// TwinCAT 3 PLC project Untitled1
// ProgramVersion: 3.1.4023.0
// libraries:
//   CmpBitmapPool, * (System)
//   Tc2_SerialCom, * (Beckhoff Automation GmbH)
//   Tc2_Standard, * (Beckhoff Automation GmbH)
//   Tc2_SUPS, * (Beckhoff Automation GmbH)
//   Tc2_System, * (Beckhoff Automation GmbH)
//   Tc2_Utilities, * (Beckhoff Automation GmbH)
//   Tc3_Module, * (Beckhoff Automation GmbH)
//   VisuDialogs, * (System)
//   VisuSymbols,3.5.10.0,System
// project tree:
//   01. MAIN/01.1 ReactorTemperature/DUTs/ ST_PidParameters.TcDUT
//   01. MAIN/01.1 ReactorTemperature/FBs/ FB_PidControllerRelayOutput.TcPOU, FB_ReactorTemperatureControlStateMachine.TcPOU (not stored)
//   01. MAIN/01.1 ReactorTemperature/Handlers/01.1.1 TemperatureSensorScaling/ TemperatureSensorScalingHandler.TcPOU
//   01. MAIN/01.1 ReactorTemperature/Handlers/01.1.2 ReactorTemperatureControl/ ReactorTemperatureControlHandler.TcPOU
//   01. MAIN/01.1 ReactorTemperature/ ReactorTemperatureController.TcPOU
//   01. MAIN/01.2 ReactorLevelAndPressure/DUTs/ E_AutomaticExtractionState.TcDUT (not stored), ST_AutomaticExtractionParameters.TcDUT (not stored), ST_AutomaticExtractionValues.TcDUT, ST_ExtractiveControlValveCommands.TcDUT, ST_ExtractiveControlValveParameters.TcDUT, ST_ExtractiveOnOffValveValues.TcDUT (not stored), ST_PressureIntervals.TcDUT (not stored)
//   01. MAIN/01.2 ReactorLevelAndPressure/FBs/ FB_AutomaticExtractionStateMachine.TcPOU, FB_ControlValveStateMachine.TcPOU, FB_ExtractiveOutletControl.TcPOU, FB_ReactorValves.TcPOU, FB_Runtime.TcPOU, FB_ValveTrigger.TcPOU (not stored), F_RoundToClosest.TcPOU (not stored)
//   01. MAIN/01.2 ReactorLevelAndPressure/Handlers/01.2.1 PressureSensorScaling/ PressureSensorScalingHandler.TcPOU
//   01. MAIN/01.2 ReactorLevelAndPressure/Handlers/01.2.2 AutomaticExtraction/ AutomaticExtractionHandler.TcPOU
//   01. MAIN/01.2 ReactorLevelAndPressure/Handlers/01.2.3 ExtractiveOutlet/ ExtractiveOutletHandler.TcPOU
//   01. MAIN/01.2 ReactorLevelAndPressure/ ReactorLevelAndPressureController.TcPOU
//   01. MAIN/01.3 ReactorFlow/DUTs/ ST_FlowControlCommands.TcDUT, ST_FlowControlParameters.TcDUT, ST_MPC_Matrices.TcDUT
//   01. MAIN/01.3 ReactorFlow/FBs/ FB_ConsumptionCalculator.TcPOU, FB_mF.TcPOU, FB_MovingAverage.TcPOU, FB_MPC.TcPOU
//   01. MAIN/01.3 ReactorFlow/Handlers/01.3.1 Co2MeanFlowCalculation/ FB_Co2MeanFlowCalculationHandler.TcPOU
//   01. MAIN/01.3 ReactorFlow/Handlers/01.3.2 Co2Consumption/ FB_Co2ConsumptionHandler.TcPOU
//   01. MAIN/01.3 ReactorFlow/Handlers/01.3.3 Co2FlowModeling/ FB_Co2FlowModelingHandler.TcPOU
//   01. MAIN/01.3 ReactorFlow/Handlers/01.3.4 Co2FlowModelDeviation/ FB_Co2FlowModelDeviationHandler.TcPOU
//   01. MAIN/01.3 ReactorFlow/Handlers/01.3.5 FlowMpc/ FB_FlowMpcHandler.TcPOU
//   01. MAIN/01.3 ReactorFlow/ ReactorFlowController.TcPOU
//   01. MAIN/01.4 DataAcquisition/ DataAcquisitionController.TcPOU
//   01. MAIN/01.4 DataAcquisition/DUTs/ ST_MatlabValues.TcDUT (not stored)
//   01. MAIN/01.4 DataAcquisition/FBs/ FB_HeartBeat.TcPOU
//   01. MAIN/01.4 DataAcquisition/Handlers/01.4.1 OpcTagWriting/ OpcTagWritingHandler.TcPOU
//   01. MAIN/01.4 DataAcquisition/Handlers/01.4.2 Matlab/ MatlabHandler.TcPOU (not stored)
//   01. MAIN/01.4 DataAcquisition/Handlers/01.4.3 SpecialDataWriting/ SpecialDataWritingHandler.TcPOU
//   01. MAIN/01.6 VariablePersistence/ VariablePersistenceController.TcPOU
//   01. MAIN/01.5 SerialCommunication/DUTs/ ST_SerialCommReadData.TcDUT, ST_SerialCommSetpoints.TcDUT (not stored)
//   01. MAIN/01.5 SerialCommunication/FBs/ FB_SerialCom.TcPOU, FB_UpdateSetpoint.TcPOU
//   01. MAIN/01.5 SerialCommunication/FUNs/ F_AsciiNumberConvert.TcPOU, F_NumberAsciiConvert.TcPOU (not stored)
//   01. MAIN/01.5 SerialCommunication/Handlers/01.5.1 SerialData/ SerialDataHandler.TcPOU
//   01. MAIN/01.5 SerialCommunication/ SerialCommunicationController.TcPOU
//   01. MAIN/01.7 Safety/Handlers/01.6.1 UiEstop/ UiEstopHandler.TcPOU (not stored)
//   01. MAIN/01.7 Safety/ SafetyController.TcPOU (not stored)
//   01. MAIN/Common/FBs/ FB_StateSpaceModel.TcPOU, FB_ToggleHeartBeat.TcPOU
//   01. MAIN/Common/FUNs/ F_AnalogScale.TcPOU
//   01. MAIN/Common/ITFs/ I_PidController.TcIO
//   01. MAIN/ MAIN.TcPOU
//   02. MAIN_Fast/02.1 BackgroundEL/ BackgroundElController.TcPOU
//   02. MAIN_Fast/ MAIN_Fast.TcPOU
//   03. VISUs/03.02 Process View/ ProcessViewBindings.TcPOU, ProcessView.TcVIS
//   03. VISUs/03.03 Parameter View/ ParameterView.TcVIS, ParameterViewBindings.TcPOU
//   03. VISUs/03.01 MainScreen View/ MainScreenBindings.TcPOU, MainScreen.TcVIS
//   03. VISUs/User Controls/ Valve.TcVIS, ValveDiagonal.TcVIS
//   05. Simulation/05.01 SimulationView/ SimulationView.TcVIS, SimulationViewBindings.TcPOU
//   05. Simulation/ Simulation.TcPOU
//   / GlobalTextList.TcGTLO, PlcTask.TcTTO, PlcTaskFast.TcTTO, Visualization Manager.TcVMO (not stored), VISU_TASK.TcTTO (not stored)
//   04. GVLs/ GVL_OPC.TcGVL, GVL_Serial.TcGVL (not stored), GVL_IO.TcGVL
//   Trash/AutoExtractionParameterMenu View/ AutoExtractionParameterMenu.TcVIS (not stored), AutoExtractionParameterMenuBindings.TcPOU (not stored)
//   Trash/ExtractiveOutletValveParameterMenu/ ExtractiveOutletValveParameterMenu.TcVIS, ExtractiveOutletValveParameterMenuBindings.TcPOU
//   Trash/ FB_PIDrelayOutput.TcPOU (not stored), LevelControlParamMenu.TcVIS (excluded from build), MainScreen_1.TcVIS (excluded from build), MainScreen_OLD.TcVIS (excluded from build), ReadWriteOPCvariables.TcPOU (excluded from build), RunMATLAB.TcPOU (not stored) (excluded from build), SerialCommunicationHandler_1.TcPOU (not stored) (excluded from build), SerialCommVisuTest.TcVIS (excluded from build), SerialCommVisuTest_1.TcVIS (excluded from build), ST_MainScreenBindingsOutputs.TcDUT (excluded from build)
//   Trash/PidParameterMenu View/ PidParameterMenu.TcVIS (not stored), PidParameterMenuBindings.TcPOU (not stored)
//   Trash/PressureAndLevelControl/ ReactorLevelAndPressureControl.TcPOU (not stored) (excluded from build), reactorpresslevelvanhaVARA.TcPOU (not stored) (excluded from build)
//   Trash/TemperatureControl/ ReactorTemperatureControl.TcPOU (not stored) (excluded from build)
//   Trash/TemperatureControl/vanhat/ FB_TemperaturePIDControl.TcPOU, TemperatureControl.TcPOU
//   Trash/TemperatureControl/vanhat/FUNs/ F_ContactorControl.TcPOU, F_GetPIDOntime.TcPOU (not stored), F_PercentageToTime.TcPOU (not stored)
//   Trash/TemperatureControl/vanhat/LevelControl/ FB_LevelControl.TcPOU (not stored), FB_LimitSwitch.TcPOU, LevelControl.TcPOU
//   Trash/TemperatureControl/vanhat/PressureControl/ FB_PIDsetpointOutput.TcPOU, PressureControl.TcPOU
//   03. VISUs/ ImagePool.TcIPO (not stored)
// real-time tasks:
//   TASK PlcTask: cycle T#10ms, priority 20, ADS port 350
//   TASK VISU_TASK: cycle T#200000us, priority 30, ADS port 351
//   TASK PlcTaskFast: cycle T#2ms, priority 1, ADS port 352
//   TASK PlcTask1: cycle T#10ms, priority 21, ADS port 353
// I/O:
//   DEVICE Device 1 (EtherCAT), AmsNetId 5.86.83.4.2.1
//     Term 1 (EK1200) [EK1200-5000 EtherCAT Power supply (2A E-Bus)]
//       Term 3 (EL2008)
//       Term 11 (EL3204) [EL3204 4Ch. Ana. Input PT100 (RTD)]
//       Term 6 (EL6021) [EL6021 Interface (RS422/485)]
//       Term 5 (EL1004) [EL1004 4Ch. Dig. Input 24V, 3ms]
//       Term 14 (EL3154) [EL3154 4Ch. Ana. Input 4-20mA]
//       Term 8 (EL9011) [EL9011 End Terminal]
// variable links:
//   Untitled1/Untitled1 Instance <-> Device 1 (EtherCAT)/Term 1 (EK1200)/Term 11 (EL3204)
//     PlcTask Inputs/GVL_IO.reactorTemperatureLower <-> RTD Inputs Channel 2/Reactor lower temperature
//     PlcTask Inputs/GVL_IO.reactorTemperatureUpper <-> RTD Inputs Channel 1/Reactor upper temperature
//   Untitled1/Untitled1 Instance <-> Device 1 (EtherCAT)/Term 1 (EK1200)/Term 14 (EL3154)
//     PlcTask Inputs/GVL_IO.reactorPressure <-> AI Standard Channel 1/Reactor pressure
//   Untitled1/Untitled1 Instance <-> Device 1 (EtherCAT)/Term 1 (EK1200)/Term 3 (EL2008)
//     PlcTask Outputs/GVL_IO.extractiveOutletControlValveClose <-> Channel 5/Extractive outlet control valve close button
//     PlcTask Outputs/GVL_IO.extractiveOutletControlValveOpen <-> Channel 4/Extractive outlet control valve open button
//     PlcTask Outputs/GVL_IO.extractiveOutletOnOffValve <-> Channel 6/Extractive outlet on/off valve button
//     PlcTask Outputs/GVL_IO.reactorInletValve <-> Channel 2/Slurry inlet valve
//     PlcTask Outputs/GVL_IO.reactorOutletValve <-> Channel 3/Slurry outlet valve
//     PlcTask Outputs/GVL_IO.reactorTemperatureContactor <-> Channel 1/Reactor temperature contactor
//   Untitled1/Untitled1 Instance <-> Device 1 (EtherCAT)/Term 1 (EK1200)/Term 5 (EL1004)
//     PlcTask Inputs/GVL_IO.reactorLevelHigh <-> Channel 2/Reactor high level
//     PlcTask Inputs/GVL_IO.reactorLevelLow <-> Channel 1/Reactor low level
//   Untitled1/Untitled1 Instance <-> Device 1 (EtherCAT)/Term 1 (EK1200)/Term 6 (EL6021)
//     PlcTaskFast Inputs/BackgroundElController.stIn_EL6001/D <-> COM TxPDO-Map Inputs/Data In 0
//     PlcTaskFast Inputs/BackgroundElController.stIn_EL6001/D @bit {8..168 step 8} <-> COM TxPDO-Map Inputs/Data In {1..21}  (21 links)
//     PlcTaskFast Inputs/BackgroundElController.stIn_EL6001/Status <-> COM TxPDO-Map Inputs/Status
//     PlcTaskFast Outputs/BackgroundElController.stOut_EL6001/Ctrl <-> COM RxPDO-Map Outputs/Ctrl
//     PlcTaskFast Outputs/BackgroundElController.stOut_EL6001/D <-> COM RxPDO-Map Outputs/Data Out 0
//     PlcTaskFast Outputs/BackgroundElController.stOut_EL6001/D @bit {8..168 step 8} <-> COM RxPDO-Map Outputs/Data Out {1..21}  (21 links)

CONFIGURATION Untitled1
    RESOURCE PLC ON TwinCAT3
        TASK PlcTask(INTERVAL := T#10ms, PRIORITY := 20);
        TASK PlcTaskFast(INTERVAL := T#2ms, PRIORITY := 1);
        PROGRAM MAIN WITH PlcTask : MAIN;
        PROGRAM MAIN_Fast WITH PlcTaskFast : MAIN_Fast;
    END_RESOURCE
END_CONFIGURATION

// ---- 01. MAIN/01.1 ReactorTemperature/DUTs/ST_PidParameters.TcDUT
TYPE ST_PidParameters :
STRUCT
	Iterationtime: REAL;
	PB: REAL;
	Ti: REAL;
	Td: REAL;
	Bias: REAL;
END_STRUCT
END_TYPE

// ---- 01. MAIN/01.2 ReactorLevelAndPressure/DUTs/ST_AutomaticExtractionValues.TcDUT
TYPE ST_AutomaticExtractionValues :
STRUCT
	elapsedTime : TIME;
	currentTimer : TIME;
	timeVisible : BOOL;
END_STRUCT
END_TYPE

// ---- 01. MAIN/01.2 ReactorLevelAndPressure/DUTs/ST_ExtractiveControlValveCommands.TcDUT
TYPE ST_ExtractiveControlValveCommands :
STRUCT
	openPercentage : DINT;
	calibrate : BOOL;
	stopCalibration : BOOL;
	requireCalibration : BOOL;
END_STRUCT
END_TYPE

// ---- 01. MAIN/01.2 ReactorLevelAndPressure/DUTs/ST_ExtractiveControlValveParameters.TcDUT
TYPE ST_ExtractiveControlValveParameters :
STRUCT
	timeToFullyOpenMs : DINT;
	calibrationTimeMs : DINT;
END_STRUCT
END_TYPE

// ---- 01. MAIN/01.3 ReactorFlow/DUTs/ST_FlowControlCommands.TcDUT
TYPE ST_FlowControlCommands :
STRUCT
	resetCo2Consumption : BOOL;
	startMovingAvgCalculation : BOOL;
	enableFlowMpc : BOOL;
	flowSetpoint : REAL;
END_STRUCT
END_TYPE

// ---- 01. MAIN/01.3 ReactorFlow/DUTs/ST_FlowControlParameters.TcDUT
TYPE ST_FlowControlParameters :
STRUCT
	movingAvgDurationSecs : INT;
	movingAvgShiftIntervalSecs : INT;
	co2ConsumptionLimit : DINT;
	excludeValuesPreFirstWindow : BOOL;
	startConsumptionCalculationWithAvg : BOOL;
	closeOnOffValveIfConsumptionExceeded : BOOL;
END_STRUCT
END_TYPE

// ---- 01. MAIN/01.3 ReactorFlow/DUTs/ST_MPC_Matrices.TcDUT
TYPE ST_MPC_Matrices :
STRUCT

gMPC_F : ARRAY[1..80,1..2] OF LREAL := [-10.110286651796301,-0.494890603179854,-9.998121030930005,-0.849211680989655,-9.882750302704293,-1.186962702093454,-9.764412993557139,-1.508607889096049,-9.643339387385019,-1.814603927230396,-9.519751705206597,-2.105399926086415,-9.393864283415191,-2.381437389289509,-9.265883750536544,-2.643150191797635,-9.136009202413343,-2.890964564494386,-9.004432375742766,-3.125299085763932,-8.871337819898013,-3.346564679742028,-8.736903066969232,-3.555164620945482,-8.601298799963665,-3.751494544990575,-8.464689019109006,-3.935942465118846,-8.327231206208078,-4.108888794256542,-8.189076486996795,-4.270706372341670,-8.050369791461257,-4.421760498660247,-7.911250012073411,-4.562408968940717,-7.771850159908285,-4.693002116962906,-7.632297518609167,-4.813882860445012,-7.492713796170435,-4.925386750979278,-7.353215274510816,-5.027842027793848,-7.213912956812981,-5.121569675125206,-7.074912712608209,-5.206883482992225,-6.936315420587746,-5.284090111169452,-6.798217109125122,-5.353489156163644,-6.660709094496298,-5.415373221003946,-6.523878116787006,-5.470027987662182,-6.387806473478991,-5.517732291925894,-6.252572150709208,-5.558758200552590,-6.118248952198138,-5.593371090539552,-5.984906625845532,-5.621829730349168,-5.852610987993847,-5.644386362935353,-5.721424045361585,-5.661286790422041,-5.591404114650545,-5.672770460290053,-5.462605939832695,-5.679070552933828,-5.335080807124128,-5.680414070454595,-5.208876657655004,-5.677021926561531,-5.084038197846002,-5.669109037457247,-4.960607007503111,-5.656884413588728,-4.838621645644044,-5.640551252149455,-4.718117754070727,-5.620307030222870,-4.599128158703624,-5.596343598461867,-4.481682968694686,-5.568847275203118,-4.365809673336917,-5.537998940919341,-4.251533236789419,-5.503974132916622,-4.138876190637855,-5.466943140187845,-4.027858724311060,-5.427071098337199,-3.918498773375450,-5.384518084494419,-3.810812105729573,-5.339439212141119,-3.704812405721946,-5.291984725775094,-3.600511356215944,-5.242300095341919,-3.497918718626178,-5.190526110366582,-3.397042410951305,-5.136798973721058,-3.297888583828834,-5.081250394967001,-3.200461694637900,-5.024007683215708,-3.104764579676458,-4.965193839450595,-3.010798524439739,-4.904927648260231,-2.918563332027186,-4.843323768932860,-2.828057389705369,-4.780492825865994,-2.739277733654720,-4.716541498247395,-2.652220111928128,-4.651572608966215,-2.566879045649682,-4.585685212715626,-2.483247888482003,-4.518974683250643,-2.401318884390793,-4.451532799767123,-2.321083223735317,-4.383447832370266,-2.242531097713636,-4.314804626603001,-2.165651751191477,-4.245684687006818,-2.090433533943659,-4.176166259689603,-2.016863950337000,-4.106324413877013,-1.944929707483633,-4.036231122425738,-1.874616761893596,-3.965955341278977,-1.805910364655540,-3.895563087846006,-1.738795105174264,-3.825117518289602,-1.673254953493765,-3.754679003706576,-1.609273301234286,-3.684305205188315,-1.546833001171776,-3.614051147749725,-1.485916405487980,-3.543969293116387,-1.426505402719236,-3.474109611361183,-1.368581453431838,-3.404519651382967];

gMPC_Phi : ARRAY[1..80,1..5] OF LREAL := [0.000284731809204,0.000000000000000,0.000000000000000,0.000000000000000,0.000000000000000,0.000363650992320,0.000284731809204,0.000000000000000,0.000000000000000,0.000000000000000,0.000438735836864,0.000363650992320,0.000284731809204,0.000000000000000,0.000000000000000,0.000510096292665,0.000438735836864,0.000363650992320,0.000284731809204,0.000000000000000,0.000577840450081,0.000510096292665,0.000438735836864,0.000363650992320,0.000284731809204,0.000642074534315,0.000577840450081,0.000510096292665,0.000438735836864,0.000363650992320,0.000702902901532,0.000642074534315,0.000577840450081,0.000510096292665,0.000438735836864,0.000760428036683,0.000702902901532,0.000642074534315,0.000577840450081,0.000510096292665,0.000814750552970,0.000760428036683,0.000702902901532,0.000642074534315,0.000577840450081,0.000865969192870,0.000814750552970,0.000760428036683,0.000702902901532,0.000642074534315,0.000914180830659,0.000865969192870,0.000814750552970,0.000760428036683,0.000702902901532,0.000959480476359,0.000914180830659,0.000865969192870,0.000814750552970,0.000760428036683,0.001001961281039,0.000959480476359,0.000914180830659,0.000865969192870,0.000814750552970,0.001041714543414,0.001001961281039,0.000959480476359,0.000914180830659,0.000865969192870,0.001078829717667,0.001041714543414,0.001001961281039,0.000959480476359,0.000914180830659,0.001113394422447,0.001078829717667,0.001041714543414,0.001001961281039,0.000959480476359,0.001145494450968,0.001113394422447,0.001078829717667,0.001041714543414,0.001001961281039,0.001175213782158,0.001145494450968,0.001113394422447,0.001078829717667,0.001041714543414,0.001202634592808,0.001175213782158,0.001145494450968,0.001113394422447,0.001078829717667,0.001227837270652,0.001202634592808,0.001175213782158,0.001145494450968,0.001113394422447,0.001250900428343,0.001227837270652,0.001202634592808,0.001175213782158,0.001145494450968,0.001271900918255,0.001250900428343,0.001227837270652,0.001202634592808,0.001175213782158,0.001290913848076,0.001271900918255,0.001250900428343,0.001227837270652,0.001202634592808,0.001308012597137,0.001290913848076,0.001271900918255,0.001250900428343,0.001227837270652,0.001323268833433,0.001308012597137,0.001290913848076,0.001271900918255,0.001250900428343,0.001336752531291,0.001323268833433,0.001308012597137,0.001290913848076,0.001271900918255,0.001348531989636,0.001336752531291,0.001323268833433,0.001308012597137,0.001290913848076,0.001358673850824,0.001348531989636,0.001336752531291,0.001323268833433,0.001308012597137,0.001367243119992,0.001358673850824,0.001348531989636,0.001336752531291,0.001323268833433,0.001374303184885,0.001367243119992,0.001358673850824,0.001348531989636,0.001336752531291,0.001379915836137,0.001374303184885,0.001367243119992,0.001358673850824,0.001348531989636,0.001384141287944,0.001379915836137,0.001374303184885,0.001367243119992,0.001358673850824,0.001387038199120,0.001384141287944,0.001379915836137,0.001374303184885,0.001367243119992,0.001388663694486,0.001387038199120,0.001384141287944,0.001379915836137,0.001374303184885,0.001389073386559,0.001388663694486,0.001387038199120,0.001384141287944,0.001379915836137,0.001388321397523,0.001389073386559,0.001388663694486,0.001387038199120,0.001384141287944,0.001386460381438,0.001388321397523,0.001389073386559,0.001388663694486,0.001387038199120,0.001383541546658,0.001386460381438,0.001388321397523,0.001389073386559,0.001388663694486,0.001379614678446,0.001383541546658,0.001386460381438,0.001388321397523,0.001389073386559,0.001374728161734,0.001379614678446,0.001383541546658,0.001386460381438,0.001388321397523,0.001368929004028,0.001374728161734,0.001379614678446,0.001383541546658,0.001386460381438,0.001362262858415,0.001368929004028,0.001374728161734,0.001379614678446,0.001383541546658,0.001354774046651,0.001362262858415,0.001368929004028,0.001374728161734,0.001379614678446,0.001346505582319,0.001354774046651,0.001362262858415,0.001368929004028,0.001374728161734,0.001337499194019,0.001346505582319,0.001354774046651,0.001362262858415,0.001368929004028,0.001327795348584,0.001337499194019,0.001346505582319,0.001354774046651,0.001362262858415,0.001317433274283,0.001327795348584,0.001337499194019,0.001346505582319,0.001354774046651,0.001306450984019,0.001317433274283,0.001327795348584,0.001337499194019,0.001346505582319,0.001294885298478,0.001306450984019,0.001317433274283,0.001327795348584,0.001337499194019,0.001282771869224,0.001294885298478,0.001306450984019,0.001317433274283,0.001327795348584,0.001270145201725,0.001282771869224,0.001294885298478,0.001306450984019,0.001317433274283,0.001257038678288,0.001270145201725,0.001282771869224,0.001294885298478,0.001306450984019,0.001243484580891,0.001257038678288,0.001270145201725,0.001282771869224,0.001294885298478,0.001229514113902,0.001243484580891,0.001257038678288,0.001270145201725,0.001282771869224,0.001215157426662,0.001229514113902,0.001243484580891,0.001257038678288,0.001270145201725,0.001200443635928,0.001215157426662,0.001229514113902,0.001243484580891,0.001257038678288,0.001185400848160,0.001200443635928,0.001215157426662,0.001229514113902,0.001243484580891,0.001170056181640,0.001185400848160,0.001200443635928,0.001215157426662,0.001229514113902,0.001154435788415,0.001170056181640,0.001185400848160,0.001200443635928,0.001215157426662,0.001138564876053,0.001154435788415,0.001170056181640,0.001185400848160,0.001200443635928,0.001122467729202,0.001138564876053,0.001154435788415,0.001170056181640,0.001185400848160,0.001106167730938,0.001122467729202,0.001138564876053,0.001154435788415,0.001170056181640,0.001089687383906,0.001106167730938,0.001122467729202,0.001138564876053,0.001154435788415,0.001073048331234,0.001089687383906,0.001106167730938,0.001122467729202,0.001138564876053,0.001056271377220,0.001073048331234,0.001089687383906,0.001106167730938,0.001122467729202,0.001039376507782,0.001056271377220,0.001073048331234,0.001089687383906,0.001106167730938,0.001022382910662,0.001039376507782,0.001056271377220,0.001073048331234,0.001089687383906,0.001005308995392,0.001022382910662,0.001039376507782,0.001056271377220,0.001073048331234,0.000988172412995,0.001005308995392,0.001022382910662,0.001039376507782,0.001056271377220,0.000970990075431,0.000988172412995,0.001005308995392,0.001022382910662,0.001039376507782,0.000953778174787,0.000970990075431,0.000988172412995,0.001005308995392,0.001022382910662,0.000936552202191,0.000953778174787,0.000970990075431,0.000988172412995,0.001005308995392,0.000919326966460,0.000936552202191,0.000953778174787,0.000970990075431,0.000988172412995,0.000902116612475,0.000919326966460,0.000936552202191,0.000953778174787,0.000970990075431,0.000884934639276,0.000902116612475,0.000919326966460,0.000936552202191,0.000953778174787,0.000867793917884,0.000884934639276,0.000902116612475,0.000919326966460,0.000936552202191,0.000850706708831,0.000867793917884,0.000884934639276,0.000902116612475,0.000919326966460,0.000833684679424,0.000850706708831,0.000867793917884,0.000884934639276,0.000902116612475,0.000816738920703,0.000833684679424,0.000850706708831,0.000867793917884,0.000884934639276,0.000799879964135,0.000816738920703,0.000833684679424,0.000850706708831,0.000867793917884];

gMPC_H : ARRAY[1..5,1..5] OF LREAL := [0.100103441989350,0.000103049987228,0.000102562271107,0.000101983140310,0.000101316783413,0.000103049987228,0.100102802181393,0.000102396694129,0.000101895423436,0.000101302677058,0.000102562271107,0.000102396694129,0.100102135118928,0.000101715791404,0.000101200618157,0.000101983140310,0.000101895423436,0.000101715791404,0.100101440088783,0.000101006570254,0.000101316783413,0.000101302677058,0.000101200618157,0.000101006570254,0.100100716386879];

gMPC_Hinv : ARRAY[1..5,1..5] OF LREAL := [9.989708039134626,-0.010252853623071,-0.010204228986415,-0.010146517228794,-0.010080136701021,-0.010252853623071,9.989771834240116,-0.010187763658072,-0.010137837465101,-0.010078817456107,-0.010204228986415,-0.010187763658072,9.989838247748814,-0.010120019713281,-0.010068756213402,-0.010146517228794,-0.010137837465101,-0.010120019713281,9.989907351206504,-0.010049549695518,-0.010080136701021,-0.010078817456107,-0.010068756213402,-0.010049549695518,9.989979217213653];

END_STRUCT
END_TYPE

// ---- 01. MAIN/01.5 SerialCommunication/DUTs/ST_SerialCommReadData.TcDUT
TYPE ST_SerialCommReadData :
STRUCT
	pumpingPressureMeasurement : DINT;
	pumpingPressureSetpoint	: DINT;
	pumpingPressureOutputPower : DINT;
	flowMeasurement : REAL;
	preHeaterTemperatureMeasurement : DINT;
	preHeaterTemperatureSetpoint : DINT;
	preHeaterTemperatureOutputPower : DINT;
	separatorTemperatureMeasurement : DINT;
	separatorTemperatureSetpoint : DINT;
	separatorTemperatureOutputPower : DINT;
END_STRUCT
END_TYPE

// ---- Trash/ST_MainScreenBindingsOutputs.TcDUT
TYPE ST_MainScreenBindingsOutputs :
STRUCT
	autoControlSelected : BOOL;// ReactorTemperatureController.autoControlSelected
	temperatureSetpoint : DINT; //ReactorTemperature.temperatureSetpoint
	manualControlPercentage : DINT;// ReactorTemperature.manualControlPercentage
	MatlabBtn : BOOL;//RunMATLAB.MatlabBtn
	OPC_ProgramNamePrefix : STRING;//GVL_OPC.OPC_ProgramNamePrefix
	StartAutomaticExtraction : BOOL;//ReactorLevelAndPressure.StartAutomaticExtraction
	estopButtonPressed : BOOL;; //Safety.buttonPressed
	estopResetPressed : BOOL; //Safety.resetPressed
	serialCommSetpoints : ST_SerialCommSetpoints;// SerialCommunicationController.SerialCommSetpoints
	
	// ProcessViewBindings in
	GVL_IO.reactorOutletValve
	GVL_IO.reactorInletValve
	ReactorTemperatureController.lowerTemperature
	ReactorTemperatureController.upperTemperature
	GVL_IO.reactorTemperatureContactor
	GVL_IO.reactorLevelHigh
	GVL_IO.reactorLevelLow
	ReactorLevelAndPressureController.iPressureScaledValue
	SerialCommunicationController.SerialCommReadData
	ReactorLevelAndPressureController.ExtractiveOnOffValveValues
	ReactorLevelAndPressureController.CalibrateDone
	ReactorLevelAndPressureController.ControlValveOpening
	ReactorLevelAndPressureController.automaticExtractionState
	SafetyController.stop

	
	// ProcessViewBindings out
	ReactorTemperatureController.temperatureContactorCommand
	ReactorLevelAndPressureController.SlurryInValveCommand
	ReactorLevelAndPressureController.PressureIntervals
	ReactorLevelAndPressureController.SlurryOutValveCommand
	ReactorLevelAndPressureController.ExtractiveOutOnOffValveCommand
	ExtractiveOutletValveCommands.calibrate
	ReactorLevelAndPressureController.ExtractiveControlValveCommands
	
	//Parametersettingsbindings in
	
	// parametersettings out
	ReactorTemperatureController.pidControllerParameters
	ReactorLevelAndPressureController.AutomaticExtractionParameters
	ReactorLevelAndPressureController.PressureIntervals
	ReactorLevelAndPressureController.ExtractiveControlValveParameters
END_STRUCT
END_TYPE

// ---- 04. GVLs/GVL_OPC.TcGVL
{attribute 'qualified_only'}
VAR_GLOBAL
	
	{attribute 'OPC.UA.DA' := '1'} OPC_TemperatureContactor : BOOL; // Temperature contactor
	{attribute 'OPC.UA.DA' := '1'} OPC_ReactorTemperature : INT; // Reactor temperature
	{attribute 'OPC.UA.DA' := '1'} OPC_ReactorLowerTemperature : INT; // Reactor temperature
	{attribute 'OPC.UA.DA' := '1'} OPC_ReactorPressure : INT; // Reactor pressure
	{attribute 'OPC.UA.DA' := '1'} OPC_ReactorTemperatureSetpoint: INT; // Reactr temperature setpoint
	{attribute 'OPC.UA.DA' := '1'} OPC_SlurryInletValve: BOOL;
	{attribute 'OPC.UA.DA' := '1'} OPC_SlurryOutletValve: BOOL;
	{attribute 'OPC.UA.DA' := '1'} OPC_ExtractiveOutletOnOffValve: BOOL;
	{attribute 'OPC.UA.DA' := '1'} OPC_ExtractiveControlValveOpening: INT;
	
	{attribute 'OPC.UA.DA' := '1'} OPC_PumpingPressure: DINT;
	{attribute 'OPC.UA.DA' := '1'} OPC_PumpingPressureSetpoint: DINT;
	
	{attribute 'OPC.UA.DA' := '1'} OPC_PreHeaterTemperature: DINT;
	{attribute 'OPC.UA.DA' := '1'} OPC_PreHeaterTemperatureSetpoint: DINT;
	
	{attribute 'OPC.UA.DA' := '1'} OPC_SeparatorTemperature: DINT;
	{attribute 'OPC.UA.DA' := '1'} OPC_SeparatorTemperatureSetpoint: DINT;
	
	{attribute 'OPC.UA.DA' := '1'} OPC_CO2VolumetricFlow: REAL;
	
	{attribute 'OPC.UA.DA' := '1'} OPC_AutoExtractionState: STRING;
	
	// Program name 
	{attribute 'OPC.UA.DA' := '1'} OPC_ProgramNamePrefix: STRING;
	
	// Special data 
	{attribute 'OPC.UA.DA' := '1'} OPC_OutletValveOpenArray: ARRAY[0..99] OF BOOL;
	{attribute 'OPC.UA.DA' := '1'} OPC_OutletValveOpenTimeStampArray: ARRAY[0..99] OF STRING;
	{attribute 'OPC.UA.DA' := '1'} OPC_OutletValveCloseArray: ARRAY[0..99] OF BOOL;
	{attribute 'OPC.UA.DA' := '1'} OPC_OutletValveCloseTimeStampArray: ARRAY[0..99] OF STRING;
END_VAR

// ---- 04. GVLs/GVL_IO.TcGVL
{attribute 'qualified_only'}
VAR_GLOBAL

	reactorTemperatureContactor AT %Q* : BOOL; // Temperature contactor
	reactorTemperatureUpper AT %I*: INT; // Reactor temperature
	reactorTemperatureLower AT %I*: INT; // Reactor temperature lower
	reactorLevelHigherHigh AT %I*: BOOL; // Higher high slurry level
	reactorLevelLow AT %I*: BOOL; // Low slurry level
	reactorLevelHigh AT %I*: BOOL; // High slurry level
	reactorLevelLowerLow AT %I*: BOOL; // Lower low slurry level
	reactorOutletValve AT %Q*: BOOL;  // Reactor outlet valve
	reactorPressure AT %I*: INT; // Reactor pressure raw analog value
	reactorInletValve AT %Q*: BOOL; // Filling valve
	extractiveOutletOnOffValve AT %Q* : BOOL;
	extractiveOutletControlValveOpen AT %Q* : BOOL;
	extractiveOutletControlValveClose AT %Q* : BOOL;
	
END_VAR

// ---- 01. MAIN/Common/ITFs/I_PidController.TcIO
INTERFACE I_PidController

METHOD AutomaticControl : BOOL
VAR_INPUT
	processVariable		: REAL; // Temperature measurement
	setpoint			: REAL; // Temperature setpoint
END_VAR
END_METHOD

METHOD ManualControl : BOOL
VAR_INPUT
	iControlPercentage : INT;
END_VAR
END_METHOD

METHOD ResetControl : BOOL
END_METHOD

METHOD SetParameters : BOOL
VAR_INPUT
	parameters			: ST_PidParameters;
END_VAR
END_METHOD

END_INTERFACE

// ---- 01. MAIN/MAIN.TcPOU
PROGRAM MAIN


(*** CONTROLLERS: MAIN LOGIC MODULARIZED ***)

// Reactor temperature
ReactorTemperatureController(
						temperatureUpper := GVL_IO.reactorTemperatureUpper,
						temperatureLower := GVL_IO.reactorTemperatureLower,
						contactor => GVL_IO.reactorTemperatureContactor);

// Reactor level/pressure
ReactorLevelAndPressureController(
					serialCommData := SerialCommunicationController.SerialCommReadData,
					stop := SafetyController.stop,
					levelHigh := GVL_IO.reactorLevelHigh,
					co2ConsumptionLimitExceeded :=  ReactorFlowController._closeOnOffValve,
					modeledValvePosition := ReactorFlowController.ModeledValvePercentage,
					flowMpcEnabled :=  ProcessViewBindings.FlowControlCommands.enableFlowMpc,
					slurryInletValve => GVL_IO.reactorInletValve,
					slurryOutletValve => GVL_IO.reactorOutletValve,
					extractiveOutletOnOffValve => GVL_IO.extractiveOutletOnOffValve,
					extractiveOutletControlValveClose => GVL_IO.extractiveOutletControlValveClose,
					extractiveOutletControlValveOpen => GVL_IO.extractiveOutletControlValveOpen);
					
// Reactor flow
ReactorFlowController(
					serialCommData := SerialCommunicationController.SerialCommReadData,
					flowControlValveOpening := ReactorLevelAndPressureController.ControlValveOpening,
					serialCommReadData := SerialCommunicationController.SerialCommReadData);
					
// Data acquisition
DataAcquisitionController(
					slurryOutletValveOpen := GVL_IO.reactorOutletValve,
					automaticExtractionStateActive := ReactorLevelAndPressureController.automaticExtractionState = E_AutomaticExtractionState.FILLING_ACTIVE);

{IF NOT defined (Simulation)}
// Persistent data saving
VariablePersistenceController();
{END_IF}

// Serial communication
SerialCommunicationController();

// Safety
SafetyController();

(*** VISUALIZATION BINDINGS: DATA TRANSFER FROM/TO UI ***)

// MainScreen in
MainScreenBindings(
				matlabValues := DataAcquisitionController.MatlabHmiValues,
				SerialCommReadData := SerialCommunicationController.SerialCommReadData,
				CalibrateDone := ReactorLevelAndPressureController.CalibrateDone,
				Stop :=  SafetyController.stop,
				ReactorPressure := ReactorLevelAndPressureController.iPressureScaledValue,
				OnOffValvePressureLimit := ParameterViewBindings.onOffValvePressureLimit);
// MainScreen out
ReactorTemperatureController.autoControlSelected := MainScreenBindings.autoControlSelected;
ReactorTemperatureController.temperatureSetpoint := MainScreenBindings.temperatureSetpoint;
ReactorTemperatureController.manualControlPercentage := MainScreenBindings.temperaturePidManualControlPercentage;
DataAcquisitionController.MatlabBtn := MainScreenBindings.matlabBtn;
GVL_OPC.OPC_ProgramNamePrefix := MainScreenBindings.programNamePrefix;
ReactorLevelAndPressureController.StartAutomaticExtraction := MainScreenBindings.startAutomaticExtraction;
SafetyController.buttonPressed := MainScreenBindings.estopButtonPressed;
SafetyController.resetPressed := MainScreenBindings.estopResetPressed;
SerialCommunicationController.SerialCommSetpoints := MainScreenBindings.serialCommSetpoints;
	
//ProcessView in			
ProcessViewBindings(
				reactorOutletValve := GVL_IO.reactorOutletValve,
				reactorInletValve := GVL_IO.reactorInletValve,
				lowerTemperature := ReactorTemperatureController.lowerTemperature,
				upperTemperature := ReactorTemperatureController.upperTemperature,
				reactorTemperatureContactor := GVL_IO.reactorTemperatureContactor,
				reactorLevelHigh := GVL_IO.reactorLevelHigh,
				reactorLevelLow := GVL_IO.reactorLevelLow,
				iPressureScaledValue := ReactorLevelAndPressureController.iPressureScaledValue,
				SerialCommReadData := SerialCommunicationController.SerialCommReadData,
				ExtractiveOnOffValveValues := ReactorLevelAndPressureController.ExtractiveOnOffValveValues,
				CalibrateDone := ReactorLevelAndPressureController.CalibrateDone,
				ControlValveOpening := ReactorLevelAndPressureController.ControlValveOpening,
				automaticExtractionState := ReactorLevelAndPressureController.automaticExtractionState,
				stop := SafetyController.stop,
				onOffValvePressureLimit := ParameterViewBindings.onOffValvePressureLimit,
				AutomaticExtractionValues := ReactorLevelAndPressureController.AutomaticExtractionValues,
				MeanReactorFlow := ReactorFlowController.MeanReactorFlow,
				ConsumedCo2Value := ReactorFlowController.ConsumedCo2Amount,
				FlowControlParameters := ParameterViewBindings.flowControlParameters,
				co2ConsumptionLimitExceeded := ReactorFlowController.Co2ConsumptionLimitExceeded,
				closeOnOffValve := ReactorFlowController.CloseOnOffValve,
				modeledMeanReactorFlow := ReactorFlowController.ModeledMeanReactorFlow,
				co2FlowDeviationPercentage := ReactorFlowController.FlowModelDeviationPercentage);
// ProcessView out
ReactorTemperatureController.temperatureContactorCommand := ProcessViewBindings.temperatureContactorCommand;
ReactorLevelAndPressureController.SlurryInValveCommand := ProcessViewBindings.SlurryInValveCommand;
ReactorLevelAndPressureController.PressureIntervals := ProcessViewBindings.PressureIntervals;
ReactorLevelAndPressureController.SlurryOutValveCommand := ProcessViewBindings.SlurryOutValveCommand;
ReactorLevelAndPressureController.ExtractiveOutOnOffValveCommand := ProcessViewBindings.ExtractiveOutOnOffValveCommand;
ReactorLevelAndPressureController.ExtractiveControlValveCommands := ProcessViewBindings.ExtractiveControlValveCommands;
ReactorFlowController.FlowControlParameters := ParameterViewBindings.flowControlParameters;
ReactorFlowController.FlowControlCommands := ProcessViewBindings.FlowControlCommands;
	
// ParameterView in			
ParameterViewBindings();
// ParameterView out
ReactorTemperatureController.pidControllerParameters := ParameterViewBindings.reactorTemperaturePidParameters;
ReactorLevelAndPressureController.AutomaticExtractionParameters := ParameterViewBindings.autoExtractionParameters;
ReactorLevelAndPressureController.PressureIntervals := ParameterViewBindings.pressureIntervals;
ReactorLevelAndPressureController.ExtractiveControlValveParameters := ParameterViewBindings.extractionValveParameters;


// Simulation
{IF defined (Simulation)}
	Simulation();
{END_IF}

END_PROGRAM

// ---- 01. MAIN/01.1 ReactorTemperature/ReactorTemperatureController.TcPOU
PROGRAM ReactorTemperatureController
VAR_INPUT
	temperatureUpper : INT;
	temperatureLower : INT;
END_VAR
VAR_OUTPUT
	contactor : BOOL;
END_VAR
VAR
	
	// Handlers to call
	HandleTemperatureSensorScaling : TemperatureSensorScalingHandler;
	HandleReactorTemperatureControl : ReactorTemperatureControlHandler;
	
	// Internal variables
	_pidControllerParameters : ST_PidParameters;
	_manualControlPercentage : INT;
	_upperTemperature : INT;
	_lowerTemperature : INT;
	_temperatureSetpoint : INT;
	_temperatureContactor : BOOL;
	_autoControlSelected : BOOL;
	_temperatureContactorCommand : BOOL;
END_VAR


HandleTemperatureSensorScaling(
						upperTemperatureSensor := GVL_IO.reactorTemperatureUpper,
						lowerTemperatureSensor := GVL_IO.reactorTemperatureLower,
						upperTemperatureValue => _upperTemperature,
						lowerTemperatureValue => _lowerTemperature);
						
HandleReactorTemperatureControl(
						pidControllerParameters := _pidControllerParameters,
						manualControlPercentage := _manualControlPercentage,
						upperTemperature := _upperTemperature,
						lowerTemperature := _lowerTemperature,
						temperatureSetpoint := _temperatureSetpoint,
						autoControlSelected := _autoControlSelected,
						temperatureContactorCommand := _temperatureContactorCommand ,
						temperatureContactor => contactor);

PROPERTY autoControlSelected : BOOL
SET

_autoControlSelected := autoControlSelected;
END_SET
END_PROPERTY

PROPERTY lowerTemperature : INT
GET

lowerTemperature := _lowerTemperature;
END_GET
END_PROPERTY

PROPERTY manualControlPercentage : INT
SET


_manualControlPercentage := manualControlPercentage;
END_SET
END_PROPERTY

PROPERTY pidControllerParameters : ST_PidParameters
SET

_pidControllerParameters := pidControllerParameters;
END_SET
END_PROPERTY

PROPERTY temperatureContactor : BOOL
GET

temperatureContactor := _temperatureContactor;
END_GET
END_PROPERTY

PROPERTY temperatureContactorCommand : BOOL
SET

_temperatureContactorCommand := temperatureContactorCommand;
END_SET
END_PROPERTY

PROPERTY temperatureSetpoint : INT
SET

_temperatureSetpoint := temperatureSetpoint;
END_SET
END_PROPERTY

PROPERTY upperTemperature : INT
GET

upperTemperature := _upperTemperature;
END_GET
END_PROPERTY

END_PROGRAM

// ---- 01. MAIN/01.1 ReactorTemperature/Handlers/01.1.1 TemperatureSensorScaling/TemperatureSensorScalingHandler.TcPOU
FUNCTION_BLOCK TemperatureSensorScalingHandler
VAR_INPUT
	upperTemperatureSensor : INT;
	lowerTemperatureSensor : INT;
END_VAR
VAR_OUTPUT
	upperTemperatureValue : INT;
	lowerTemperatureValue : INT;
END_VAR
VAR
END_VAR


upperTemperatureValue	:= upperTemperatureSensor/10;
lowerTemperatureValue := lowerTemperatureSensor/10;

END_FUNCTION_BLOCK

// ---- 01. MAIN/01.1 ReactorTemperature/Handlers/01.1.2 ReactorTemperatureControl/ReactorTemperatureControlHandler.TcPOU
FUNCTION_BLOCK ReactorTemperatureControlHandler
VAR_INPUT
	pidControllerParameters : ST_PidParameters;
	manualControlPercentage : INT;
	upperTemperature : INT;
	lowerTemperature : INT;
	temperatureSetpoint : INT;
	autoControlSelected : BOOL;
	temperatureContactorCommand : BOOL;
END_VAR
VAR_OUTPUT
	temperatureContactor : BOOL;
END_VAR
VAR
	TemperatureControlStateMachine : FB_ReactorTemperatureControlStateMachine;
END_VAR

TemperatureControlStateMachine(temperatureMeasurement := TO_REAL(upperTemperature),
							temperatureSetpoint := TO_REAL(temperatureSetpoint),
							pidParameters := pidControllerParameters,
							manualControlPercentage := manualControlPercentage,
							autoControlSelected := autoControlSelected,
							relayOn => temperatureContactor);

IF autoControlSelected OR (NOT autoControlSelected AND manualControlPercentage > 0) THEN
	temperatureContactor := TemperatureControlStateMachine.relayOn;
ELSE
	temperatureContactor := temperatureContactorCommand;
END_IF

END_FUNCTION_BLOCK

// ---- 01. MAIN/01.2 ReactorLevelAndPressure/ReactorLevelAndPressureController.TcPOU
PROGRAM ReactorLevelAndPressureController
VAR_INPUT
	serialCommData : ST_SerialCommReadData;
	stop : BOOL;
	levelHigh : BOOL;
	co2ConsumptionLimitExceeded : BOOL;
	modeledValvePosition : DINT;
	flowMpcEnabled : BOOL;
END_VAR
VAR_OUTPUT
	slurryInletValve : BOOL;
	slurryOutletValve : BOOL;
	extractiveOutletOnOffValve : BOOL;
	extractiveOutletControlValveClose : BOOL;
	extractiveOutletControlValveOpen : BOOL;
END_VAR
VAR
	
	// Handlers to call
	HandlePressureSensorScaling : PressureSensorScalingHandler;
	HandleAutomaticExtraction : AutomaticExtractionHandler;
	HandleExtractiveOutlet : ExtractiveOutletHandler;

	_iPressureScaledValue: INT; //Scaled pressure value
	_bLevelControlSwitch : BOOL;
	_slurryInValveCommand : BOOL;
	_slurryOutValveCommand : BOOL;
	_pressureIntervals : ST_PressureIntervals;
	_extractiveControlValveCommands : ST_ExtractiveControlValveCommands;
	_ExtractiveControlValveParameters : ST_ExtractiveControlValveParameters;
	_automaticExtractionParameters : ST_AutomaticExtractionParameters;
	_decreasePumpSetpoint : BOOL;
	_controlValveOpening : DINT;
	_calibrateDone : BOOL;
	
	_extractiveOutOnOffValveCommand : BOOL;
	_startAutomaticExtraction : BOOL;
	
	_automaticExtractionState : E_AutomaticExtractionState;
	_automaticExtractionValues : ST_AutomaticExtractionValues;
	_extractiveOnOffValveValues : ST_ExtractiveOnOffValveValues;
END_VAR
VAR PERSISTENT
	_fillingValveOpenInterval: INT;
	_fillingValveCloseInterval: INT;	
END_VAR


HandlePressureSensorScaling(
						reactorPressureSensor := GVL_IO.reactorPressure,
						PressureScaledValue => _iPressureScaledValue);

HandleAutomaticExtraction(
						automaticExtractionParameters := _automaticExtractionParameters,
						extractiveControlValveParameters := _extractiveControlValveParameters,
						pressureScaledValue := _iPressureScaledValue,
						serialCommData := serialCommData,
						extractiveControlValveCommands := _extractiveControlValveCommands,
						pressureIntervals := _pressureIntervals,
						reactorLevelHigh := levelHigh,
						startAutomaticExtraction := _startAutomaticExtraction,
						calibrateDone := _calibrateDone,
						slurryInValveCommand := _slurryInValveCommand,
						slurryOutValveCommand := _slurryOutValveCommand,
						decreasePumpSetpoint => _decreasePumpSetpoint,
						reactorInletValve => slurryInletValve,
						automaticExtractionState => _automaticExtractionState,
						extractiveOutOnOffValveAutoCommand => ,
						controlValveAutoOpenPercentage => ,
						reactorOutletValve => slurryOutletValve,
						automaticExtractionValues => _automaticExtractionValues);
						
HandleExtractiveOutlet(
					stop := stop,
					extractiveControlValveCommands := _ExtractiveControlValveCommands,
					extractiveControlValveParameters := _ExtractiveControlValveParameters,
					extractiveOutOnOffValveCommand := (_extractiveOutOnOffValveCommand AND (_automaticExtractionState = E_AutomaticExtractionState.MANUAL_EXTRACTION)) OR 
														((_automaticExtractionState <> E_AutomaticExtractionState.MANUAL_EXTRACTION) AND HandleAutomaticExtraction.extractiveOutOnOffValveAutoCommand AND NOT co2ConsumptionLimitExceeded),
					autoExtractionControlValveValue := HandleAutomaticExtraction.controlValveAutoOpenPercentage,
					autoExtractionStarted := _automaticExtractionState <> E_AutomaticExtractionState.MANUAL_EXTRACTION,
					modeledValvePosition := modeledValvePosition,
					flowMpcEnabled := flowMpcEnabled,
					controlValveOpeningPercentage => _controlValveOpening,
					extractiveOnOffValveValues => _extractiveOnOffValveValues,
					calibrateDone => _calibrateDone,
					openOnOffValve => extractiveOutletOnOffValve,
					closeExtractiveOutletValve => extractiveOutletControlValveClose,
					openExtractiveOutletValve => extractiveOutletControlValveOpen);

//IF _startAutomaticExtraction AND _calibrateDone THEN
//	manualModeEntered := FALSE;
	
//	// Automatic extraction
//	AutomaticExtraction(
//				parameters := _automaticExtractionParameters,
//				controlValveFullOpenTime := _ExtractiveControlValveParameters.timeToFullyOpenMs,
//				reactorPressure := _iPressureScaledValue,
//				pumpPressure := serialCommData.pumpingPressureMeasurement,
//				pumpSetpoint := SerialCommData.pumpingPressureSetpoint,
//				decreasePumpSetpoint => _decreasePumpSetpoint,
//				extractivePumpOn => GVL_IO.reactorInletValve,
//				co2onOffValveClosed => ,
//				automaticExtractionState => _automaticExtractionState);
//	_extractiveOutOnOffValveCommand := NOT AutomaticExtraction.co2onOffValveClosed;
//	_extractiveControlValveCommands.openPercentage := AutomaticExtraction.controlValveOpeningPercentage;
	
//	// Slurry outlet valve control
//	RTRIG_SetPressureReference(CLK := _automaticExtractionState = E_AutomaticExtractionState.FILLING_ACTIVE);
//	IF RTRIG_SetPressureReference.Q THEN
//		pressureReference :=  _iPressureScaledValue;
//	END_IF
//	SlurryOutValveControl.pressureIntervalControl(
//										interval_1_condition:= GVL_IO.reactorInletValve,// GVL_IO.reactorLevelHigh AND GVL_IO.reactorInletValve, // If above higher limit and filling valve open
//										pressureUpperInterval_1:= _pressureIntervals.PressureUpperInterval_1, 
//										pressureLowerInterval_1:= _pressureIntervals.PressureLowerInterval_1, 
//										interval_2_condition:= FALSE,//GVL_IO.reactorLevelHigh AND NOT GVL_IO.reactorInletValve,  // If above higher limit and filling valve closed
//										pressureUpperInterval_2:= _pressureIntervals.PressureUpperInterval_2, 
//										pressureLowerInterval_2:= _pressureIntervals.PressureLowerInterval_2, 
//										interval_3_condition:= FALSE,//NOT GVL_IO.reactorLevelHigh AND GVL_IO.reactorInletValve,  // If below higher limit and reactor filling valve open
//										pressureUpperInterval_3:= _pressureIntervals.PressureUpperInterval_3, 
//										pressureLowerInterval_3:= _pressureIntervals.PressureLowerInterval_3, 
//										pressureValue:= _iPressureScaledValue,  
//										pressureReference:= pressureReference,//_iPressureScaledValue,//DINT_TO_INT(SerialCommunicationHandler.pumpingPressureSetpoint), 
//										valveOpenCondition:= NOT (NOT GVL_IO.reactorLevelHigh AND NOT GVL_IO.reactorInletValve), 
//										forceValveClosed:= (NOT GVL_IO.reactorLevelHigh AND NOT GVL_IO.reactorInletValve),
//										);
//	GVL_IO.reactorOutletValve := SlurryOutValveControl.pressureControlOpen;
	
//ELSE
//	AutomaticExtraction.resetState();
//	// Close inlet/outlet valves when manual mode entered
//	IF NOT manualModeEntered THEN
//		GVL_IO.reactorInletValve := FALSE; // Close all valves when auto mode is exited
//		GVL_IO.reactorOutletValve := FALSE;
//		autoModeEntered := FALSE;
//		manualModeEntered := TRUE;
//	END_IF
//	GVL_IO.reactorInletValve := _slurryInValveCommand;
//	GVL_IO.reactorOutletValve := _slurryOutValveCommand;

//	_automaticExtractionState := E_AutomaticExtractionState.MANUAL_EXTRACTION;
	
//END_IF

//// Extractive outlet control
//_extractiveControlValveCommands.stopCalibration := Safety.stop;
//HandleExtractiveOutlet(
//					onOffValveCommand := _extractiveOutOnOffValveCommand,
//					controlValveCommands := _ExtractiveControlValveCommands,
//					controlValveParameters := _ExtractiveControlValveParameters,
//					onOffValveOpen => ,
//					onOffValveButtonCommand => GVL_IO.extractiveOutletOnOffValve,
//					controlValveClose => GVL_IO.extractiveOutletControlValveClose,
//					controlValveOpen => GVL_IO.extractiveOutletControlValveOpen,
//					controlValveCurrentOpenPercentage => _controlValveOpening,
//					calibrateDone => _calibrateDone);
//_extractiveOnOffValveValues.open := HandleExtractiveOutlet.onOffValveOpen;

PROPERTY AutomaticExtractionParameters : ST_AutomaticExtractionParameters
SET

_automaticExtractionParameters := AutomaticExtractionParameters;
END_SET
END_PROPERTY

PROPERTY automaticExtractionState : E_AutomaticExtractionState
GET

automaticExtractionState := _automaticExtractionSTate;
END_GET
END_PROPERTY

PROPERTY AutomaticExtractionValues : ST_AutomaticExtractionValues
GET

AutomaticExtractionValues := _automaticExtractionValues;
END_GET
END_PROPERTY

PROPERTY bLevelControlSwitch : BOOL
SET

_bLevelControlSwitch := bLevelControlSwitch;
END_SET
END_PROPERTY

PROPERTY CalibrateDone : BOOL
GET

CalibrateDone := _calibrateDone;
END_GET
END_PROPERTY

PROPERTY ControlValveOpening : DINT
GET

ControlValveOpening := _controlValveOpening;
END_GET
END_PROPERTY

PROPERTY controlValveOpeningOrClosing : BOOL
GET

controlValveOpeningOrClosing := GVL_IO.extractiveOutletControlValveClose OR GVL_IO.extractiveOutletControlValveOpen;
END_GET
END_PROPERTY

PROPERTY decreasePumpSetpoint : BOOL
GET

decreasePumpSetpoint := _decreasePumpSetpoint;
END_GET
END_PROPERTY

PROPERTY ExtractiveControlValveCommands : ST_ExtractiveControlValveCommands
SET
IF NOT _startAutomaticExtraction THEN
	_ExtractiveControlValveCommands := ExtractiveControlValveCommands;
END_IF
END_SET
END_PROPERTY

PROPERTY ExtractiveControlValveParameters : ST_ExtractiveControlValveParameters
SET

_ExtractiveControlValveParameters := ExtractiveControlValveParameters;
END_SET
END_PROPERTY

PROPERTY ExtractiveOnOffValveValues : ST_ExtractiveOnOffValveValues
GET

ExtractiveOnOffValveValues := _extractiveOnOffValveValues;
END_GET
END_PROPERTY

PROPERTY ExtractiveOutOnOffValveCommand : BOOL
SET

_extractiveOutOnOffValveCommand := ExtractiveOutOnOffValveCommand;
END_SET
END_PROPERTY

PROPERTY fillingValveCloseInterval : INT
SET

_fillingValveCloseInterval := fillingValveCloseInterval;
END_SET
END_PROPERTY

PROPERTY fillingValveOpenInterval : INT
SET

_fillingValveOpenInterval := fillingValveOpenInterval;
END_SET
END_PROPERTY

PROPERTY iPressureScaledValue : INT
GET

iPressureScaledValue := _iPressureScaledValue;
END_GET
END_PROPERTY

PROPERTY PressureIntervals : ST_PressureIntervals
SET

_pressureIntervals := PressureIntervals;
END_SET
END_PROPERTY

PROPERTY SlurryInValveCommand : BOOL
SET

_slurryInValveCommand := SlurryInValveCommand;
END_SET
END_PROPERTY

PROPERTY SlurryOutValveCommand : BOOL
SET

_slurryOutValveCommand := SlurryOutValveCommand;
END_SET
END_PROPERTY

PROPERTY StartAutomaticExtraction : BOOL
SET

_startAutomaticExtraction := StartAutomaticExtraction;
END_SET
END_PROPERTY

END_PROGRAM

// ---- 01. MAIN/01.2 ReactorLevelAndPressure/Handlers/01.2.1 PressureSensorScaling/PressureSensorScalingHandler.TcPOU
FUNCTION_BLOCK PressureSensorScalingHandler
VAR_INPUT
	reactorPressureSensor : INT;
END_VAR
VAR_OUTPUT
	PressureScaledValue : INT;
END_VAR
VAR
END_VAR


// Scale analog pressure
PressureScaledValue := F_AnalogScale(AnalogInputRawValue := reactorPressureSensor, MaxAnalogValue := 1000);

END_FUNCTION_BLOCK

// ---- 01. MAIN/Common/FUNs/F_AnalogScale.TcPOU
FUNCTION F_AnalogScale : INT
VAR_INPUT
	AnalogInputRawValue	: DINT;
	MaxAnalogValue		: INT;
END_VAR
VAR
	MaxInput			: INT;
	ScaledValue: INT;
END_VAR
VAR_OUTPUT
END_VAR

// 4-20 mA: 0-32767
MaxInput := 32767;
F_AnalogScale := REAL_TO_INT(AnalogInputRawValue / (MaxInput / MaxAnalogValue));

END_FUNCTION

// ---- 01. MAIN/01.2 ReactorLevelAndPressure/Handlers/01.2.2 AutomaticExtraction/AutomaticExtractionHandler.TcPOU
FUNCTION_BLOCK AutomaticExtractionHandler
VAR_INPUT
	automaticExtractionParameters : ST_AutomaticExtractionParameters;
	extractiveControlValveParameters : ST_ExtractiveControlValveParameters;	
	pressureScaledValue: INT; //Scaled pressure value 
	serialCommData : ST_SerialCommReadData;
	extractiveControlValveCommands : ST_ExtractiveControlValveCommands;
	pressureIntervals : ST_PressureIntervals;
	reactorLevelHigh : BOOL;
	startAutomaticExtraction : BOOL;
	calibrateDone : BOOL;
	slurryInValveCommand : BOOL;
	slurryOutValveCommand : BOOL;
END_VAR
VAR_OUTPUT
	decreasePumpSetpoint : BOOL;
	reactorInletValve : BOOL;
	automaticExtractionState : E_AutomaticExtractionState;
	extractiveOutOnOffValveAutoCommand : BOOL;
	reactorOutletValve : BOOL;
	controlValveAutoOpenPercentage : DINT;
	automaticExtractionValues : ST_AutomaticExtractionValues;
END_VAR
VAR
	manualModeEntered : BOOL;
	autoModeEntered : BOOL;
	SlurryOutValveControl: FB_ReactorValves;
	AutomaticExtraction : FB_AutomaticExtractionStateMachine;
	RTRIG_SetPressureReference : R_TRIG;
	pressureReference : INT;
END_VAR

IF startAutomaticExtraction AND calibrateDone THEN
	manualModeEntered := FALSE;
	
	// Automatic extraction
	AutomaticExtraction(
				parameters := automaticExtractionParameters,
				controlValveFullOpenTime := extractiveControlValveParameters.timeToFullyOpenMs,
				reactorPressure := pressureScaledValue,
				pumpPressure := serialCommData.pumpingPressureMeasurement,
				pumpSetpoint := SerialCommData.pumpingPressureSetpoint,
				decreasePumpSetpoint => decreasePumpSetpoint,
				extractivePumpOn => reactorInletValve,
				co2onOffValveClosed => ,
				automaticExtractionState => automaticExtractionState,
				automaticExtractionValues => automaticExtractionValues);
	extractiveOutOnOffValveAutoCommand := NOT AutomaticExtraction.co2onOffValveClosed;
	controlValveAutoOpenPercentage := AutomaticExtraction.controlValveOpeningPercentage;
	
	// Slurry outlet valve control
	RTRIG_SetPressureReference(CLK := automaticExtractionState = E_AutomaticExtractionState.FILLING_ACTIVE);
	IF RTRIG_SetPressureReference.Q THEN
		pressureReference :=  pressureScaledValue;
	END_IF
	IF automaticExtractionState = E_AutomaticExtractionState.FILLING_ACTIVE THEN
		SlurryOutValveControl.pressureIntervalControl(
											interval_1_condition:= reactorInletValve,// GVL_IO.reactorLevelHigh AND GVL_IO.reactorInletValve, // If above higher limit and filling valve open
											pressureUpperInterval_1:= pressureIntervals.PressureUpperInterval_1, 
											pressureLowerInterval_1:= pressureIntervals.PressureLowerInterval_1, 
											interval_2_condition:= FALSE,//GVL_IO.reactorLevelHigh AND NOT GVL_IO.reactorInletValve,  // If above higher limit and filling valve closed
											pressureUpperInterval_2:= pressureIntervals.PressureUpperInterval_2, 
											pressureLowerInterval_2:= pressureIntervals.PressureLowerInterval_2, 
											interval_3_condition:= FALSE,//NOT GVL_IO.reactorLevelHigh AND GVL_IO.reactorInletValve,  // If below higher limit and reactor filling valve open
											pressureUpperInterval_3:= pressureIntervals.PressureUpperInterval_3, 
											pressureLowerInterval_3:= pressureIntervals.PressureLowerInterval_3, 
											pressureValue:= pressureScaledValue,  
											pressureReference:= pressureReference,//_iPressureScaledValue,//DINT_TO_INT(SerialCommunicationHandler.pumpingPressureSetpoint), 
											valveOpenCondition:=  automaticExtractionState = E_AutomaticExtractionState.FILLING_ACTIVE,//NOT (NOT reactorLevelHigh AND NOT reactorInletValve), 
											forceValveClosed:= FALSE,//(NOT reactorLevelHigh AND NOT reactorInletValve),
											);
		reactorOutletValve := SlurryOutValveControl.pressureControlOpen;
	ELSE 
		reactorOutletValve := FALSE;
	END_IF
	
ELSE
	AutomaticExtraction.resetState();
	decreasePumpSetpoint := FALSE;
	// Close inlet/outlet valves when manual mode entered
	IF NOT manualModeEntered THEN
		reactorInletValve := FALSE; // Close all valves when auto mode is exited
		reactorOutletValve := FALSE;
		autoModeEntered := FALSE;
		manualModeEntered := TRUE;
	END_IF
	reactorInletValve := slurryInValveCommand;
	reactorOutletValve := slurryOutValveCommand;

	automaticExtractionState := E_AutomaticExtractionState.MANUAL_EXTRACTION;
	automaticExtractionValues.timeVisible := FALSE;
	
END_IF

automaticExtraction.getCurrentTimer();

END_FUNCTION_BLOCK

// ---- 01. MAIN/01.2 ReactorLevelAndPressure/FBs/FB_ReactorValves.TcPOU
FUNCTION_BLOCK FB_ReactorValves
VAR_INPUT
END_VAR
VAR_OUTPUT
	pressureControlOpen : BOOL; // Valve to control via pressure intervals
	timeControlOpen : BOOL; // Valve to control via on/off time intervals
END_VAR
VAR
	timeControlToggle: FB_ToggleHeartBeat;
	openInterval : INT;
	closeInterval : INT;
END_VAR

METHOD onOffTimeControl : BOOL
VAR_INPUT
	openIntervalSecs : INT; // Time for valve to stay open
	closeIntervalSecs : INT; // Time for valve to stay closed
END_VAR

openInterval := openIntervalSecs;
closeInterval := closeIntervalSecs ;
timeControlToggle(I_OpenInterValSecs := openInterval, I_CloseIntervalSecs := closeInterval, O_Update => timeControlOpen);
END_METHOD

METHOD pressureIntervalControl : BOOL
VAR_INPUT
	interval_1_condition: BOOL; // Condition for applying intervals marked with 1
	pressureUpperInterval_1 : INT;
	pressureLowerInterval_1 : INT;
	interval_2_condition: BOOL; // Condition for applying intervals marked with 2
	pressureUpperInterval_2 : INT;
	pressureLowerInterval_2 : INT;	
	interval_3_condition: BOOL; // Condition for applying intervals marked with 3
	pressureUpperInterval_3 : INT;
	pressureLowerInterval_3 : INT;	
	pressureValue : INT; // Pressure measurement
	pressureReference : INT; // Pressure reference (setpoint)
	valveOpenCondition : BOOL; // Condition for opening valve, must be filled for other factors to applu
	forceValveClosed : BOOL; // Condition for forcing valve closed independent of other factors
END_VAR

VAR
	pressureUpperInterval : INT;
	pressureLowerInterval: INT;
END_VAR

IF interval_1_condition THEN
	pressureUpperInterval := pressureUpperInterval_1;
	pressureLowerInterval := pressureLowerInterval_1;
ELSIF interval_2_condition THEN
	pressureUpperInterval := pressureUpperInterval_2;
	pressureLowerInterval := pressureLowerInterval_2;	
ELSIF interval_3_condition THEN
	pressureUpperInterval := pressureUpperInterval_3;
	pressureLowerInterval := pressureLowerInterval_3;		
END_IF

// Control valve when intervals are exceeded
IF (pressureValue >= pressureReference + pressureUpperInterval) AND valveOpenCondition THEN
	pressureControlOpen := TRUE;
ELSIF (pressureValue <= pressureReference - pressureLowerInterval) OR forceValveClosed THEN
	pressureControlOpen := FALSE;
END_IF
END_METHOD

END_FUNCTION_BLOCK

// ---- 01. MAIN/Common/FBs/FB_ToggleHeartBeat.TcPOU
FUNCTION_BLOCK FB_ToggleHeartBeat
VAR_INPUT
	I_OpenIntervalSecs : INT;
	I_CloseIntervalSecs : INT;
END_VAR
VAR_OUTPUT
	O_Update : BOOL;
END_VAR
VAR
	TON_LifeBitOff: TON;
	TON_LifeBitOn: TON;
END_VAR


TON_LifeBitOn(IN:= NOT O_Update, PT:=INT_TO_TIME(I_CloseIntervalSecs)*1000, Q=> , ET=> );
IF TON_LifeBitOn.Q THEN
	O_Update := TRUE;
END_IF
TON_LifeBitOff(IN:= O_Update , PT:=INT_TO_TIME(I_OpenIntervalSecs)*1000 , Q=>, ET=> ); 
IF TON_LifeBitOff.Q THEN
	O_Update := FALSE;
END_IF

METHOD firstTime : BOOL
VAR_INPUT
	entered : BOOL;
END_VAR

VAR
	enter: BOOL;
END_VAR
IF entered THEN
	//O_Update := TRUE;
END_IF
//IF enter THEN
	//O_Update := TRUE;
//END_IF
END_METHOD

END_FUNCTION_BLOCK

// ---- 01. MAIN/01.2 ReactorLevelAndPressure/FBs/FB_AutomaticExtractionStateMachine.TcPOU
FUNCTION_BLOCK FB_AutomaticExtractionStateMachine
VAR_INPUT
	parameters : ST_AutomaticExtractionParameters;
	controlValveFullOpenTime : DINT;
	reactorPressure : DINT;
	pumpPressure : DINT;
	pumpSetpoint : DINT;
END_VAR
VAR_OUTPUT
	controlValveOpeningPercentage : DINT;
	decreasePumpSetpoint : BOOL;
	extractivePumpOn : BOOL;
	co2onOffValveClosed : BOOL;
	fillingActive : BOOL;
	automaticExtractionState : E_AutomaticExtractionState;
	automaticExtractionValues : ST_AutomaticExtractionValues;
END_VAR
VAR
	TON_FillingTimer : TON;
	TON_WaitForValve : TON;
	TON_WaitForPressure : TON;
	TON_KeepExtractivePumpOn : TON;
	startingReactorPRessure : DINT;
	startingPumpSetpoint : DINT;
	startingPumpPressure : DINT;
	endingPumpPressure : DINT;
	TON_FillingPumpWaitTimer : TON;
	
END_VAR

CASE automaticExtractionState OF 
	
	E_AutomaticExtractionState.AUTO_EXTRACTION: // Extraction step
		IF controlValveOpeningPercentage <> parameters.controlValveOpeningValue THEN
			automaticExtractionState := 6;
		END_IF
		fillingActive := FALSE;
		// Start filling timer. When filling timer exceeded, move to filling step
		TON_FillingTimer(
						IN := TRUE,
						PT := TO_TIME(parameters.fillingTime*1000));
		IF TON_FillingTimer.Q THEN
			TON_FillingTimer(IN := FALSE);
			startingPumpSetpoint := pumpSetpoint;// Log setpoint at the moment filling procedure starts
			automaticExtractionState := automaticExtractionState + 1;
		END_IF
		
	E_AutomaticExtractionState.REDUCING_CONTROL_VALVE: // Filling step: Control valve to a small opening
		
		fillingActive := TRUE;
		controlValveOpeningPercentage := 20;
		TON_WaitForValve(
						IN := TRUE,
						PT := TO_TIME(1000));//controlValveFullOpenTime*1000));
		IF TON_WaitForValve.Q THEN
			TON_WaitForValve(IN := FALSE);
			automaticExtractionState := automaticExtractionState + 1;
		END_IF		
	E_AutomaticExtractionState.REDUCING_CO2_PUMP_SETPOINT: // Set pump setpoint to 80 bar
	
		decreasePumpSetpoint := TRUE;
//		TON_WaitForPressure(
//							IN := TRUE,
//							PT := TO_TIME(parameters.pumpSetpointWaitTime*1000));
//		IF TON_WaitForPressure.Q THEN
//			TON_WaitForPressure(IN := FALSE);
//			co2onOffValveClosed := TRUE;  // Close co2 on/off valve
//			automaticExtractionState := automaticExtractionState + 1;
//		END_IF
		IF pumpPressure <= startingPumpSetpoint THEN
			TON_WaitForPressure(IN := FALSE);
			automaticExtractionState := automaticExtractionState + 1;			
		END_IF
		
	E_AutomaticExtractionState.CLOSING_ON_OFF_VALVE:
	
		co2onOffValveClosed := TRUE;  // Close co2 on/off valve
		TON_FillingPumpWaitTimer(IN := TRUE, PT := TO_TIME(parameters.pumpWaitTime*1000));
		IF TON_FillingPumpWaitTimer.Q THEN
			TON_FillingPumpWaitTimer(IN := FALSE);
			startingReactorPressure := reactorPressure;
			startingPumpPressure := pumpPressure;
			automaticExtractionState := automaticExtractionState + 1;		
		END_IF
	
	E_AutomaticExtractionState.FILLING_ACTIVE: //  extractive pump on: stays on for a desired time
	
//		co2onOffValveClosed := TRUE;
		extractivePumpOn := TRUE;
		TON_KeepExtractivePumpOn(
								IN := TRUE,
								PT := TO_TIME(parameters.pumpOnTime*1000));
		IF TON_KeepExtractivePumpOn.Q THEN
			TON_KeepExtractivePumpOn(IN := FALSE);
			endingPumpPressure := pumpPressure;
			automaticExtractionState := automaticExtractionState + 1;
		END_IF
	
	E_AutomaticExtractionState.TURNING_EXTRACTIVE_PUMP_OFF: // Extractive pump turns off after pressure reaches the same as it was b4 turning on
	
		IF (startingReactorPRessure + (startingPumpPressure - endingPumpPressure)) <= reactorPressure THEN
			extractivePumpOn := FALSE;
			automaticExtractionState := automaticExtractionState + 1;
		END_IF
		
	E_AutomaticExtractionState.INCREASING_CO2_PUMP_SETPOINT: // Pressure setpoint back to original (+40bar) and open on/off valve
	
		co2onOffValveClosed := FALSE;
		decreasePumpSetpoint := FALSE;
		automaticExtractionState := automaticExtractionState + 1;
	
	E_AutomaticExtractionState.OPENING_CONTROL_VALVE_TO_SETPOINT: // open control valve to desired value
	
		controlValveOpeningPercentage := parameters.controlValveOpeningValue;
		automaticExtractionState := 0;
		
END_CASE

METHOD getCurrentTimer : BOOL
VAR_INPUT
END_VAR

CASE automaticExtractionState OF 
	
	E_AutomaticExtractionState.AUTO_EXTRACTION: // Extraction step

		automaticExtractionValues.currentTimer := TON_FillingTimer.PT;
		automaticExtractionValues.elapsedTime := TON_FillingTimer.ET;
		automaticExtractionValues.timeVisible := TRUE;
		
	E_AutomaticExtractionState.REDUCING_CONTROL_VALVE: // Filling step: Control valve to a small opening
		
		automaticExtractionValues.currentTimer := TON_WaitForValve.PT;
		automaticExtractionValues.elapsedTime := TON_WaitForValve.ET;
		automaticExtractionValues.timeVisible := TRUE;
	
	E_AutomaticExtractionState.REDUCING_CO2_PUMP_SETPOINT: // Set pump setpoint to 80 bar

		automaticExtractionValues.timeVisible := FALSE;	
		
	E_AutomaticExtractionState.CLOSING_ON_OFF_VALVE:
	
		automaticExtractionValues.currentTimer := TON_FillingPumpWaitTimer.PT;
		automaticExtractionValues.elapsedTime := TON_FillingPumpWaitTimer.ET;
		automaticExtractionValues.timeVisible := TRUE;

	E_AutomaticExtractionState.FILLING_ACTIVE: //  extractive pump on: stays on for a desired time
	
		automaticExtractionValues.currentTimer := TON_KeepExtractivePumpOn.PT;
		automaticExtractionValues.elapsedTime := TON_KeepExtractivePumpOn.ET;
		automaticExtractionValues.timeVisible := TRUE;
	
	E_AutomaticExtractionState.TURNING_EXTRACTIVE_PUMP_OFF: // Extractive pump turns off after pressure reaches the same as it was b4 turning on

		automaticExtractionValues.timeVisible := FALSE;	
		
	E_AutomaticExtractionState.INCREASING_CO2_PUMP_SETPOINT: // Pressure setpoint back to original (+40bar) and open on/off valve

		automaticExtractionValues.timeVisible := FALSE;	
	
	E_AutomaticExtractionState.OPENING_CONTROL_VALVE_TO_SETPOINT: // open control valve to desired value

		automaticExtractionValues.timeVisible := FALSE;	

END_CASE
END_METHOD

METHOD resetState : BOOL
VAR_INPUT
END_VAR

automaticExtractionState := 0;
TON_FillingTimer(IN :=FALSE);
TON_WaitForValve(IN :=FALSE);
TON_WaitForPressure(IN :=FALSE);
TON_KeepExtractivePumpOn(IN :=FALSE);
co2onOffValveClosed := FALSE;
decreasePumpSetpoint := FALSE;
extractivePumpOn := FALSE;
fillingActive := FALSE;
END_METHOD

END_FUNCTION_BLOCK

// ---- 01. MAIN/01.2 ReactorLevelAndPressure/Handlers/01.2.3 ExtractiveOutlet/ExtractiveOutletHandler.TcPOU
FUNCTION_BLOCK ExtractiveOutletHandler
VAR_INPUT
	stop : BOOL;
	extractiveControlValveCommands : ST_ExtractiveControlValveCommands;
	extractiveControlValveParameters : ST_ExtractiveControlValveParameters;
	extractiveOutOnOffValveCommand : BOOL;
	autoExtractionControlValveValue : DINT;
	autoExtractionStarted : BOOL;
	modeledValvePosition : DINT;
	flowMpcEnabled : BOOL;
END_VAR
VAR_OUTPUT
	extractiveOnOffValveValues : ST_ExtractiveOnOffValveValues;
	controlValveOpeningPercentage : DINT;
	calibrateDone : BOOL;
	openOnOffValve : BOOL;
	closeExtractiveOutletValve : BOOL;
	openExtractiveOutletValve : BOOL;
END_VAR
VAR
	ExtractiveOutletControl : FB_ExtractiveOutletControl;
	RTRIG_AutomaticExtractionStopped : R_TRIG;
	RTRIG_EstopPRessed : R_TRIG;
END_VAR


extractiveControlValveCommands.stopCalibration := stop;

IF autoExtractionStarted THEN
	extractiveControlValveCommands.openPercentage := autoExtractionControlValveValue;
END_IF

RTRIG_AutomaticExtractionStopped(CLK := NOT autoExtractionStarted);
RTRIG_EstopPRessed(CLK := stop);
extractiveControlValveCommands.requireCalibration := RTRIG_EstopPRessed.q;//RTRIG_AutomaticExtractionStopped.Q OR RTRIG_EstopPRessed.q;

IF flowMpcEnabled THEN
	extractiveControlValveCommands.openPercentage := modeledValvePosition;
END_IF

ExtractiveOutletControl(
					onOffValveCommand := extractiveOutOnOffValveCommand,
					controlValveCommands := extractiveControlValveCommands,
					controlValveParameters := extractiveControlValveParameters,
					onOffValveOpen => ,
					onOffValveButtonCommand => openOnOffValve,//GVL_IO.extractiveOutletOnOffValve,
					controlValveClose => closeExtractiveOutletValve,
					controlValveOpen => openExtractiveOutletValve,
					controlValveCurrentOpenPercentage => controlValveOpeningPercentage,
					calibrateDone => calibrateDone);
					
extractiveOnOffValveValues.open := ExtractiveOutletControl.onOffValveOpen;

END_FUNCTION_BLOCK

// ---- 01. MAIN/01.2 ReactorLevelAndPressure/FBs/FB_ExtractiveOutletControl.TcPOU
FUNCTION_BLOCK FB_ExtractiveOutletControl
VAR_INPUT
	onOffValveCommand : BOOL;
	controlValveCommands : ST_ExtractiveControlValveCommands;
	controlValveParameters : ST_ExtractiveControlValveParameters;
END_VAR
VAR_OUTPUT
	onOffValveOpen : BOOL;
	onOffValveButtonCommand	: BOOL;
	controlValveClose	: BOOL;
	controlValveOpen	: BOOL;
	controlValveCurrentOpenPercentage : DINT;
	calibrateDone : BOOL;
END_VAR
VAR
	TON_OpenValve : TOF;
	TON_CloseValve : TOF;
	calibrate : BOOL;
	ControlValveStateMachine : FB_ControlValveStateMachine;
	onOffValveButton : FB_ValveTrigger;
END_VAR

//onOffValveOpen := onOffValveCommand;
onOffValveButton(
			openCommand := onOffValveCommand);
onOffValveButtonCommand := onOffValveButton.buttonCommand;
onOffValveOpen := onOffValveButton.isOpen;


ControlValveStateMachine(
						controlValveCommands := controlValveCommands,
						controlValveParameters := controlValveParameters,
						closeControlValve => controlValveClose,
						openControlValve => controlValveOpen,
						currentControlValveOpenPercentage => controlValveCurrentOpenPercentage,
						calibrateDone => calibrateDone);

END_FUNCTION_BLOCK

// ---- 01. MAIN/01.2 ReactorLevelAndPressure/FBs/FB_ControlValveStateMachine.TcPOU
FUNCTION_BLOCK FB_ControlValveStateMachine
VAR_INPUT
	controlValveCommands : ST_ExtractiveControlValveCommands;
	controlValveParameters : ST_ExtractiveControlValveParameters;
END_VAR
VAR_OUTPUT
	closeControlValve : BOOL;
	openControlValve : BOOL;
	currentControlValveOpenPercentage : DINT;
	calibrateDone : BOOL;
	test : real;
END_VAR
VAR
	startCalibrate : BOOL;
	RTRIG_startCalibrate : R_TRIG;
	RTRIG_requireCalibration : R_TRIG;
	controlState : INT;
	TOF_Calibration : TOF;
	closeCommand : BOOL;
	
	openvalve : FB_Runtime;//(resetToTime := T#0S);
	closevalve : FB_Runtime;//(resetToTime := TO_TIME(controlValveParameters.timeToFullyOpenMs));
	start : BOOL;
	setvalve : BOOL;
	open : BOOL;
	close : BOOL;
END_VAR

// Read commands from ui
startCalibrate := controlValveCommands.calibrate;
RTRIG_startCalibrate(CLK := startCalibrate);
RTRIG_requireCalibration(CLK := controlValveCommands.requireCalibration);

CASE controlState OF 
	
	0: // Before calibration
		closeCommand := FALSE;
		calibrateDone := FALSE;
		IF RTRIG_startCalibrate.Q THEN
			controlState := 1;
		END_IF
	
	1: // Calibrate
		TOF_Calibration(IN := startCalibrate, PT := TO_TIME(controlValveParameters.calibrationTimeMs));
		startCalibrate := FALSE;
		closeCommand := TRUE;
		IF controlValveCommands.stopCalibration THEN
			TOF_Calibration(IN := FALSE);
			startCalibrate := FALSE;
			controlState := 0;
		END_IF
		IF NOT TOF_Calibration.Q THEN
			TOF_Calibration(IN := TRUE);
			calibrateDone := TRUE;
			openvalve.resetValues();
			closevalve.resetValues();
			closeCommand := FALSE;
			controlState := 2;
		END_IF
	
	2: // Control
		// Calculate how long control valve should open/close
		
		IF controlValveCommands.openPercentage > currentControlValveOpenPercentage THEN
			open := TRUE;
			close := FALSE;
		ELSIF controlValveCommands.openPercentage < currentControlValveOpenPercentage THEN
			open := FALSE;
			close := TRUE;
		ELSE
			open := FALSE;
			close := FALSE;
		END_IF
		openvalve(
				gotime := open, 
				settime := TO_TIME(controlValveParameters.timeToFullyOpenMs),
				resetToTime :=  T#0S,
				countdown := close, 
				elapsedtime => , elapsed => );
		closevalve(
				gotime := close, 
				settime := TO_TIME(controlValveParameters.timeToFullyOpenMs),
			 	resetToTime := TO_TIME(controlValveParameters.timeToFullyOpenMs),
				countdown := open, elapsedtime =>, 
				elapsed => );	
		
		// Monitor calibrate command, return to calibration step
		IF RTRIG_startCalibrate.Q THEN
			controlState := 1;
		END_IF	
		// Return to pre-calibration step if stop issued
		IF RTRIG_requireCalibration.Q THEN
			controlState := 0;
			close := FALSE;
			open := FALSE;
			startCalibrate := FALSE;
		END_IF


END_CASE

// Calculate valve open-% according to open timer
IF controlValveParameters.timeToFullyOpenMs > 0 THEN
	currentControlValveOpenPercentage := TO_DINT(((TIME_TO_REAL(openvalve.elapsedtime)) /(controlValveParameters.timeToFullyOpenMs)*100));// TO_DINT(TIME_TO_REAL(openvalve.elapsedtime)/100);
	test := TO_DINT(TIME_TO_REAL(openvalve.elapsedtime));
END_IF

closeControlValve := closeCommand OR close;
openControlValve := open;

END_FUNCTION_BLOCK

// ---- 01. MAIN/01.2 ReactorLevelAndPressure/FBs/FB_Runtime.TcPOU
FUNCTION_BLOCK FB_Runtime
VAR_INPUT
	gotime: BOOL;
	settime: TIME;
	countdown: BOOL; // New input
	resetToTime : TIME;
END_VAR
VAR_OUTPUT
	elapsedtime: TIME;
	elapsed: BOOL;
END_VAR
VAR
	reset: BOOL;
	_resetTOTime : TIME;
	initial : BOOL := TRUE;
	presenttime: TIME;
	lasttime: TIME;
	cycletime: TIME;

END_VAR


_resetToTime := ResetToTime; 

IF initial THEN
	elapsedtime := _resetToTime;
	initial := FALSE;
END_IF

presenttime:= TIME();
IF NOT reset THEN
(* here the test of overflow*)
	IF (lasttime > presenttime) THEN (*overflow := true*);
		lasttime:= DWORD_TO_TIME(NOT TIME_TO_DWORD(lasttime))+T#1MS;
		cycletime:= presenttime+lasttime;
	ELSE
		cycletime:= presenttime - lasttime;
	END_IF
ELSE
	elapsedtime:=_resetToTime;
	cycletime:=t#0s;
END_IF

lasttime:=presenttime;

IF gotime AND NOT countDown THEN
		elapsedtime := elapsedtime + cycletime;
ELSIF NOT gotime AND countdown THEN
	IF elapsedtime > cycletime THEN
		elapsedtime := elapsedtime - cycletime;
	ELSE
		elapsedtime := T#0S;
	END_IF
END_IF

IF settime < elapsedtime THEN
	elapsed:=TRUE;
	elapsedtime := settime;
ELSE
	elapsed:=FALSE;
END_IF

reset := FALSE;

METHOD resetValues : BOOL
reset := TRUE;
END_METHOD

END_FUNCTION_BLOCK

// ---- 01. MAIN/01.5 SerialCommunication/SerialCommunicationController.TcPOU
PROGRAM SerialCommunicationController
VAR
	// Handlers to call
	HandleSerialCommunication : SerialDataHandler;
	
	// Local variables
	_serialCommSetpoints : ST_SerialCommSetpoints;
	_serialCommReadData : ST_SerialCommReadData;
END_VAR


HandleSerialCommunication(
						setpoints := _serialCommSetpoints,
						readData => _serialCommReadData);

PROPERTY SerialCommReadData : ST_SerialCommReadData
GET

SerialCommReadData := _serialCommReadData;
END_GET
END_PROPERTY

PROPERTY SerialCommSetpoints : ST_SerialCommSetpoints
SET

_serialCommSetpoints := SerialCommSetpoints;
END_SET
END_PROPERTY

END_PROGRAM

// ---- 01. MAIN/01.5 SerialCommunication/Handlers/01.5.1 SerialData/SerialDataHandler.TcPOU
(*
Based on SerialCom_InfoSys_Sample1 (v2.0)
This sample sends and receives a string via serial communication.
Three hardware interfaces are used: Pc COM port, EL terminal, KL terminal
*)
FUNCTION_BLOCK SerialDataHandler
VAR_INPUT
	setpoints : ST_SerialCommSetpoints;
END_VAR
VAR_OUTPUT
	readData : ST_SerialCommReadData;
END_VAR
VAR
	//fbEL6001	: FB_SerialCom;
	
	fbAsciiComm: FB_SerialCom;
	

	ReceiveStep: INT;
	pumpPressureStartSend: BOOL;
	
	fbUpdatePressureSetpoint: FB_UpdateSetpoint;
	pumpingPressureMeasurement: DINT;
	pumpingPressureSetpoint: DINT;
	pumpingPressureSetSetpoint: DINT;
	pumpingPressureSetSetpointPrev: DINT;
	tonMessageUpdate: TON;
	rTrigMessageNotUpdated: R_TRIG;
	pumpingPressureOutputPower: DINT;
	flowMeasurement: DINT;
	preHeaterTemperatureMeasurement: DINT;
	preHeaterTemperatureSetpoint: DINT;
	fbUpdatePreHeaterTemperatureSetpoint: FB_UpdateSetpoint;
	preHeaterTemperatureSetSetpointPrev: DINT;
	preHeaterTemperatureStartSend: BOOL;
	separatorTemperatureMeasurement: DINT;
	separatorTemperatureSetpoint: DINT;
	fbUpdateSeparatorTemperatureSetpoint: FB_UpdateSetpoint;
	separatorTemperatureStartSend: BOOL;
	separatorTemperatureSetSetpointPrev: DINT;
	
	pumpingPressureSentSetpoint : DINT;
	
END_VAR


// Data exchange from/to terminal
fbAsciiComm(TxBuffer:=TxBufferEL, RxBuffer:=RxBufferEL);

// Receive data
ReceiveData();

// Send data
SendData();

METHOD ReceiveData : BOOL
VAR_INPUT
END_VAR

CASE ReceiveStep OF
	0: 
		// On startup: start data receiving
		//ProcessVariableRead := TRUE;
		ReceiveStep := 1;
	1:
		// Read pressure measurement from controller
		fbAsciiComm.StartSend(SendStringIn := 'L2M?*', start := TRUE);
		IF fbAsciiComm.Received THEN
			readData.pumpingPressureMeasurement := F_AsciiNumberConvert(fbAsciiComm.sReceivedString);  
			fbAsciiComm.StopSend(stop := TRUE);
			ReceiveStep := 2;
		END_IF
	2:
		// Read pressure setpoint value
		fbAsciiComm.StartSend(SendStringIn := 'L2S?*', start := TRUE);
		IF fbAsciiComm.Received THEN
			readData.pumpingPressureSetpoint := F_AsciiNumberConvert(fbAsciiComm.sReceivedString); 
			fbAsciiComm.StopSend(stop := TRUE);
			ReceiveStep := 3;
		END_IF		
	3:
		// Read pressure controller output power
		fbAsciiComm.StartSend(SendStringIn := 'L2W?*', start := TRUE);
		IF fbAsciiComm.Received THEN
			readData.pumpingPressureOutputPower := F_AsciiNumberConvert(fbAsciiComm.sReceivedString); 
			fbAsciiComm.StopSend(stop := TRUE);
			ReceiveStep := 4;
		END_IF
	4:
		// Read flow measurement from controller
		fbAsciiComm.StartSend(SendStringIn := 'L3M?*', start := TRUE);
		IF fbAsciiComm.Received THEN
			readData.flowMeasurement := F_AsciiNumberConvert(fbAsciiComm.sReceivedString); 
			readData.flowMeasurement := readData.flowMeasurement/100;
			fbAsciiComm.StopSend(stop := TRUE);
			ReceiveStep := 5;
		END_IF
	5:
		// Read preheater measurement from controller
		fbAsciiComm.StartSend(SendStringIn := 'L4M?*', start := TRUE);
		IF fbAsciiComm.Received THEN
			readData.preHeaterTemperatureMeasurement := F_AsciiNumberConvert(fbAsciiComm.sReceivedString);  
			fbAsciiComm.StopSend(stop := TRUE);
			ReceiveStep := 6;
		END_IF
	6:
		// Read preheater setpoint value
		fbAsciiComm.StartSend(SendStringIn := 'L4S?*', start := TRUE);
		IF fbAsciiComm.Received THEN
			readData.preHeaterTemperatureSetpoint := F_AsciiNumberConvert(fbAsciiComm.sReceivedString); 
			fbAsciiComm.StopSend(stop := TRUE);
			ReceiveStep := 7;
		END_IF		
	7:
		// Read preheater controller output power
		fbAsciiComm.StartSend(SendStringIn := 'L4W?*', start := TRUE);
		IF fbAsciiComm.Received THEN
			readData.preHeaterTemperatureOutputPower := F_AsciiNumberConvert(fbAsciiComm.sReceivedString); 
			fbAsciiComm.StopSend(stop := TRUE);
			ReceiveStep := 8;
		END_IF	
	8:
		// Read separator measurement from controller
		fbAsciiComm.StartSend(SendStringIn := 'L5M?*', start := TRUE);
		IF fbAsciiComm.Received THEN
			readData.separatorTemperatureMeasurement := F_AsciiNumberConvert(fbAsciiComm.sReceivedString);  
			fbAsciiComm.StopSend(stop := TRUE);
			ReceiveStep := 9;
		END_IF
	9:
		// Read separator setpoint value
		fbAsciiComm.StartSend(SendStringIn := 'L5S?*', start := TRUE);
		IF fbAsciiComm.Received THEN
			readData.separatorTemperatureSetpoint := F_AsciiNumberConvert(fbAsciiComm.sReceivedString); 
			fbAsciiComm.StopSend(stop := TRUE);
			ReceiveStep := 10;
		END_IF		
	10:
		// Read separator controller output power
		fbAsciiComm.StartSend(SendStringIn := 'L5W?*', start := TRUE);
		IF fbAsciiComm.Received THEN
			readData.separatorTemperatureOutputPower := F_AsciiNumberConvert(fbAsciiComm.sReceivedString); 
			fbAsciiComm.StopSend(stop := TRUE);
			ReceiveStep := 0;
		END_IF
			
END_CASE
tonMessageUpdate(IN:=NOT (fbAsciiComm.bStringReceived), PT := T#2S);
rTrigMessageNotUpdated(CLK := tonMessageUpdate.Q);
IF rTrigMessageNotUpdated.Q THEN
	fbAsciiComm.StopSend(stop := TRUE);
	ReceiveStep := 0;
END_IF
END_METHOD

METHOD SendData : BOOL
VAR_INPUT
END_VAR

// Stop receiving data during send
IF pumpPressureStartSend OR preHeaterTemperatureStartSend OR separatorTemperatureStartSend THEN
	ReceiveStep := 0;
END_IF

// Update pressure setpoint
IF NOT ReactorLevelAndPressureController.decreasePumpSetpoint THEN
	pumpingPressureSentSetpoint :=  setpoints.pumpingPressureSetSetpoint;
ELSE
	pumpingPressureSentSetpoint :=	81;//_serialCommSetpoints.pumpingPressureSetSetpoint - 40; // Automatic extraction control
END_IF
fbUpdatePressureSetpoint(fbAsciiComm := fbAsciiComm, 
						bStartSend := pumpPressureStartSend, sParameterCharacter := 'S', 
						iValue := pumpingPressureSentSetpoint, 
						iSlaveNo := 2);
IF pumpingPressureSentSetpoint <> pumpingPressureSetSetpointPrev THEN
	pumpPressureStartSend := TRUE;
	fbAsciiComm.StopSend(stop := TRUE);
	pumpingPressureSetSetpointPrev := pumpingPressureSentSetpoint;
END_IF

// Update preheater temperature setpoint
fbUpdatePreHeaterTemperatureSetpoint(fbAsciiComm := fbAsciiComm, 
									bStartSend := preHeaterTemperatureStartSend, 
									sParameterCharacter := 'S', 
									iValue := setpoints.preHeaterTemperatureSetSetpoint, 
									iSlaveNo := 4);
IF setpoints.preHeaterTemperatureSetSetpoint <> preHeaterTemperatureSetSetpointPrev THEN
	preHeaterTemperatureStartSend := TRUE;
	fbAsciiComm.StopSend(stop := TRUE);
	preHeaterTemperatureSetSetpointPrev := setpoints.preHeaterTemperatureSetSetpoint;
END_IF

// Update preheater temperature setpoint
fbUpdateSeparatorTemperatureSetpoint(fbAsciiComm := fbAsciiComm, 
									bStartSend := separatorTemperatureStartSend, 
									sParameterCharacter := 'S', 
									iValue := setpoints.separatorTemperatureSetSetpoint, 
									iSlaveNo := 5);
IF setpoints.separatorTemperatureSetSetpoint <> separatorTemperatureSetSetpointPrev THEN
	separatorTemperatureStartSend := TRUE;
	fbAsciiComm.StopSend(stop := TRUE);
	separatorTemperatureSetSetpointPrev := setpoints.separatorTemperatureSetSetpoint;
END_IF
END_METHOD

END_FUNCTION_BLOCK

// ---- 01. MAIN/01.5 SerialCommunication/FBs/FB_SerialCom.TcPOU
FUNCTION_BLOCK FB_SerialCom
VAR_IN_OUT
	TxBuffer	: ComBuffer;
	RxBuffer	: ComBuffer;
END_VAR
VAR
	bStart		: BOOL;
	Timer		: TON := (PT:=T#150MS);
	fbSend		: SendString;
	bSendBusy	: BOOL;
	eSendErrorID: ComError_t;

	fbReceive		: ReceiveString;
	//sReceivedString	: STRING;
	sLastReceivedString: STRING;
	bStringReceived	: BOOL;
	bReceiveBusy	: BOOL;
	bReceiveError	: BOOL;
	eReceiveErrorID	: ComError_t;
	bReceiveTimeout	: BOOL;
	nReceiveCounter	: UDINT;
	
	fTrigReceiveBusy: F_TRIG;
	rTrigSendBusy: R_TRIG;
	sSendStringIn: STRING;
	started: BOOL;
	bStartTriggered : BOOL;
	rTrigStartTriggered: R_TRIG;
	startTimer: BOOL;
	asd: BOOL;
END_VAR
VAR_INPUT
END_VAR
VAR_OUTPUT
	sReceivedString	: STRING;
	Received : BOOL;
END_VAR


// Call the send block every second to repeat the transmission.
// Also call the block as long as it is busy to finish a transmission.
rTrigStartTriggered(CLK := bStartTriggered);
IF rTrigStartTriggered.Q THEN
	startTimer := TRUE;
END_IF
Timer(IN:= startTimer );
IF Timer.Q OR fbSend.Busy THEN
	fbSend(	SendString:= sSendStringIn, // L2S#00300* set setpoint (30 celsius), L2SI* confirm,  L2M?* read temperature
			TXbuffer:= TxBuffer,
			Busy=> bSendBusy,
			Error=> );
	IF fbSend.Error <> COMERROR_NOERROR THEN
		eSendErrorID := fbSend.Error;
	END_IF
	startTimer := FALSE; (* reset timer *)
END_IF

//	Receive string data:
//	The block receives any data strings beginning with a STX ($02) and ending with an ETX ($03) character.	
fbReceive(
	Prefix:= 'L',
	Suffix:= '*',
	Timeout:= T#2s,
	ReceivedString:= sReceivedString,
	RXbuffer:= RxBuffer,
	StringReceived=> bStringReceived,
	Busy=> bReceiveBusy,
	Error=> ,
	RxTimeout=> bReceiveTimeout );
IF fbReceive.Error <> COMERROR_NOERROR THEN
	eReceiveErrorID := fbReceive.Error;
END_IF
IF bStringReceived THEN
	nReceiveCounter := nReceiveCounter + 1;
	sLastReceivedString := sReceivedString;
END_IF
fTrigReceiveBusy(CLK:=bReceiveBusy);
IF fTrigReceiveBusy.Q THEN
	Received := TRUE;
END_IF

METHOD StartSend : BOOL
VAR_INPUT
	start : BOOL;
	SendStringIn : STRING;
END_VAR

bStartTriggered := start;
sSendStringIn := SendStringIn;
END_METHOD

METHOD StopSend : BOOL
VAR_INPUT
	stop : BOOL;
END_VAR

IF stop THEN
	bstart := FALSE;
	bStartTriggered := FALSE;
	Received := FALSE;
END_IF
END_METHOD

END_FUNCTION_BLOCK

// ---- 01. MAIN/01.5 SerialCommunication/FBs/FB_UpdateSetpoint.TcPOU
FUNCTION_BLOCK FB_UpdateSetpoint
VAR_IN_OUT
	bStartSend : BOOL;	
	fbAsciiComm : FB_SerialCom;
END_VAR
VAR_INPUT
	sParameterCharacter : STRING;
	iValue				: DINT;
	iSlaveNo			: INT;
END_VAR
VAR_OUTPUT
END_VAR
VAR
	sValue: STRING;
	SendStep: INT;
	startDataSend: BOOL;
	newDataReceived: BOOL;
	startConfirmationSend: BOOL;
	ConfirmationReceived: BOOL;
	StartMsgString: STRING;
	tonMessageUpdate: TON;
	rTrigMessageNotUpdated: R_TRIG;
	ConfMsgString: STRING(255);
END_VAR

// Convert numerical value to string
sValue := F_NumberAsciiConvert(iValue);

// Compile start message string
StartMsgString := CONCAT('L',INT_TO_STRING(iSlaveNo));
StartMsgString := CONCAT(StartMsgString, sParameterCharacter);
StartMsgString := CONCAT(StartMsgString, '#');
StartMsgString := CONCAT(StartMsgString, sValue);
StartMsgString := CONCAT(StartMsgString, '0*');

// Compile confirmation message string
ConfMsgString := CONCAT('L',INT_TO_STRING(iSlaveNo));
ConfMsgString := CONCAT(ConfMsgString, sParameterCharacter);
ConfMsgString := CONCAT(ConfMsgString, 'I');
ConfMsgString := CONCAT(ConfMsgString, '*');


//fbAsciiComm(TxBuffer:=TxBufferEL, RxBuffer:=RxBufferEL);

// Send data to controller
CASE SendStep OF
	0: 
		// Wait for send command
		IF bStartSend THEN
			fbAsciiComm.StopSend(stop := TRUE);
			SendStep := 1;
		END_IF
	1:
		// Start data send
		fbAsciiComm.StartSend(SendStringIn := StartMsgString, Start := TRUE);
		IF fbAsciiComm.Received THEN
			fbAsciiComm.StopSend(stop := TRUE);
			SendStep := 2;
		END_IF
	2:
		// Send confirmation
		fbAsciiComm.StartSend(SendStringIn := ConfMsgString, Start := TRUE);
		IF fbAsciiComm.Received THEN
			fbAsciiComm.StopSend(stop := TRUE);
			bStartSend := FALSE;
			SendStep := 0;
		END_IF
	
END_CASE

tonMessageUpdate(IN:=NOT (fbAsciiComm.bStringReceived), PT := T#500MS);
rTrigMessageNotUpdated(CLK := tonMessageUpdate.Q);
IF rTrigMessageNotUpdated.Q THEN
	fbAsciiComm.StopSend(stop := TRUE);
	SendStep := 0;
END_IF

END_FUNCTION_BLOCK

// ---- 01. MAIN/01.5 SerialCommunication/FUNs/F_AsciiNumberConvert.TcPOU
FUNCTION F_AsciiNumberConvert : DINT
VAR_INPUT
	AsciiString : STRING;
END_VAR
VAR
	iValue: DINT;
	sValueString: STRING(255);
	sFirstNumber: STRING(255);
	sSecondNumber: STRING(255);
END_VAR


// Seperate number from string
sValueString := MID(AsciiString,4,4);
sFirstNumber := LEFT(sValueString,1);
sSecondNumber := LEFT(sValueString,2);
IF sFirstNumber = '0' AND sSecondNumber = '0' THEN
	iValue := STRING_TO_DINT(RIGHT(sValueString,2));
ELSIF sFirstNumber = '0' AND sSecondNumber <> '0' THEN
	iValue := STRING_TO_DINT(RIGHT(sValueString,3));
ELSE
	iValue := STRING_TO_DINT(sValueString);	
END_IF
F_AsciiNumberConvert := iValue;

END_FUNCTION

// ---- 01. MAIN/01.3 ReactorFlow/ReactorFlowController.TcPOU
PROGRAM ReactorFlowController
VAR_INPUT
	serialCommData : ST_SerialCommReadData;
	flowControlValveOpening : DINT;
	serialCommReadData : ST_SerialCommReadData;
END_VAR
VAR
	
	// Handlers to call
	HandleCo2MeanFlowCalculation : FB_Co2MeanFlowCalculationHandler;
	HandleCo2Consumption : FB_Co2consumptionHandler;
	HandleCo2FlowModeling : FB_Co2FlowModelingHandler;
	HandleCo2FlowModelDeviation : FB_Co2FlowModelDeviationHandler(maxValue := 0.35);
	HandleFlowMpc : FB_FlowMpcHandler;
	
	// Local variables
	_meanReactorFlow : REAL;
	_flowControlParameters : ST_FlowControlParameters;
	_consumedCo2Amount : REAL;
	_flowControlCommands : ST_FlowControlCommands;
	_co2ConsumptionLimitExceeded : BOOL;
	_modeledReactorMeanFlow : REAL;
	_closeOnOffValve : BOOL;
	_flowModelDeviationPercentage : DINT;
	_modeledValvePercentage : DINT;
END_VAR

HandleCo2MeanFlowCalculation(
				serialCommData := serialCommData,
				flowControlParameters := _flowControlParameters,
				startCalculation := _flowControlCommands.startMovingAvgCalculation,
				meanReactorFlow => _meanReactorFlow);
				
HandleCo2Consumption(
				meanFlow := _meanReactorFlow,
				flowControlParameters := _flowControlParameters,
				resetInput := _flowControlCommands.resetCo2Consumption,
				consumedCo2Amount => _consumedCo2Amount,
				limitExceeded => _co2ConsumptionLimitExceeded,
				closeOnOffValve => _closeOnOffValve);
				
HandleCo2FlowModeling(
				valvePositionPercentage := flowControlValveOpening,
				pumpingPressureDelta := serialCommReadData.pumpingPressureSetpoint-serialCommReadData.pumpingPressureMeasurement,
				flowMeasurement := _meanReactorFlow,
				modelingActive := _flowControlCommands.startMovingAvgCalculation,
				modeledOutput => _modeledReactorMeanFlow);
				
HandleCo2FlowModelDeviation(
				currentFlow := _meanReactorFlow,
				modeledFlow := _modeledReactorMeanFlow,
				deviationPercentage => _flowModelDeviationPercentage);
				
HandleFlowMpc(
			flowModel := HandleCo2FlowModeling.mF,
			enable := _FlowControlCommands.enableFlowMpc,
			flowSetpoint := _FlowControlCommands.flowSetpoint,
			pumpingPressureDelta := serialCommReadData.pumpingPressureSetpoint-serialCommReadData.pumpingPressureMeasurement,
			currentValvePosition := ReactorLevelAndPressureController.ControlValveOpening,
			measuredFlow := ReactorFlowController.MeanReactorFlow,
			modeledValvePercentage => _modeledValvePercentage,);

PROPERTY CloseOnOffValve : BOOL
GET

CloseOnOffValve := _closeOnOffValve;
END_GET
END_PROPERTY

PROPERTY Co2ConsumptionLimitExceeded : BOOL
GET

Co2ConsumptionLimitExceeded := _co2ConsumptionLimitExceeded;
END_GET
END_PROPERTY

PROPERTY ConsumedCo2Amount : REAL
GET

ConsumedCo2Amount := _consumedCo2Amount;
END_GET
END_PROPERTY

PROPERTY FlowControlCommands : ST_FlowControlCommands
SET

_flowControlCommands := FlowControlCommands;
END_SET
END_PROPERTY

PROPERTY FlowControlParameters : ST_FlowControlParameters
SET

_flowControlParameters := FlowControlParameters;
END_SET
END_PROPERTY

PROPERTY FlowModelDeviationPercentage : DINT
GET

FlowModelDeviationPercentage := _flowModelDeviationPercentage;
END_GET
END_PROPERTY

PROPERTY MeanReactorFlow : REAL
GET

MeanReactorFlow := _meanReactorFlow;
END_GET
END_PROPERTY

PROPERTY ModeledMeanReactorFlow : REAL
GET

ModeledMeanReactorFlow := _modeledReactorMeanFlow;
END_GET
END_PROPERTY

PROPERTY ModeledValvePercentage : DINT
GET

ModeledValvePercentage := _modeledValvePercentage;
END_GET
END_PROPERTY

END_PROGRAM

// ---- 01. MAIN/01.3 ReactorFlow/Handlers/01.3.1 Co2MeanFlowCalculation/FB_Co2MeanFlowCalculationHandler.TcPOU
FUNCTION_BLOCK FB_Co2MeanFlowCalculationHandler
VAR_INPUT
	serialCommData : ST_SerialCommReadData;
	flowControlParameters : ST_FlowControlParameters;
	startCalculation : BOOL;
END_VAR
VAR_OUTPUT
	meanReactorFlow : REAL;
END_VAR
VAR
	reactorFlow : REAL;
	flowMovingAvg : FB_MovingAverage;
	parameters : ST_FlowControlParameters;
	resetActive : BOOL;
END_VAR


reactorFlow := serialCommData.flowMeasurement;

// Calculate mean flow 
IF startCalculation THEN
	flowMovingAvg.startCalculation(
								start := TRUE,
								measurement := reactorFlow,
								windowS := flowControlParameters.movingAvgDurationSecs,
								intervalS := flowControlParameters.movingAvgShiftIntervalSecs,
								dtime := T#10MS,
								excludeUntilReady := flowControlParameters.excludeValuesPreFirstWindow);
	resetActive := FALSE;
ELSE
	IF NOT resetActive THEN
		flowMovingAvg.reset();
		resetActive := TRUE;
	END_IF
END_IF

meanReactorFlow := flowMovingAvg.value;

END_FUNCTION_BLOCK

// ---- 01. MAIN/01.3 ReactorFlow/FBs/FB_MovingAverage.TcPOU
FUNCTION_BLOCK FB_MovingAverage
VAR_OUTPUT
	ready : BOOL;
	value : REAL;
END_VAR
VAR
    sum           : REAL;
    count         : UDINT;
    running       : BOOL;
    elapsedTime   : TIME;
	
	addToSum		: BOOL;
	elapsedSecond	: INT;
	valueArray		: ARRAY[1..999] OF REAL;
	i				: INT;
	
    intervalTime : TIME;
END_VAR

METHOD reset : BOOL
VAR_INPUT
END_VAR

value := 0;
ready := FALSE;
sum := 0;
count := 0;
running := FALSE;
elapsedTime := T#0S;
elapsedSecond := 0;
FOR i := 1 TO 999 DO
	valueArray[i] := 0;
END_FOR
END_METHOD

METHOD startCalculation : BOOL
VAR_INPUT
    start : BOOL;
    measurement : REAL;
    windowS : INT;
	intervalS : INT;
    dtime : TIME;  
	excludeUntilReady : BOOL;
END_VAR

// If window is 0, return immediately
IF windowS = 0 THEN
	RETURN;
END_IF

// Start edge
IF start AND NOT running THEN
    running := TRUE;
END_IF

IF running THEN
	elapsedTime := elapsedTime + dtime;
	intervalTime := intervalTime + dtime;
	
	// Every second, calculate new mean value and shift values forward
	IF ready THEN
		IF (TIME_TO_DINT(intervalTime))/1000 >= intervalS THEN
			addToSum := TRUE;
			elapsedSecond := elapsedSecond + 1;
			FOR i := 1 TO windowS DO
				sum := sum + valueArray[i];
			END_FOR
			value := sum/windowS;
			// Shift values
			FOR i := 1 TO windowS - 1 DO
				valueArray[i] := valueArray[i + 1];
			END_FOR
			valueArray[windowS] := measurement;
			intervalTime := T#0S;
			sum := 0;
		END_IF
	ELSE
		IF (TIME_TO_DINT(intervalTime))/1000 >= intervalS THEN
			elapsedSecond := elapsedSecond + 1;
			valueArray[elapsedSecond] := measurement;
			intervalTime := T#0S;
			IF NOT excludeUntilReady THEN
				FOR i := 1 TO elapsedSecond DO
					sum := sum + valueArray[i];
				END_FOR
				value := sum / elapsedSecond;
				sum := 0;
			ELSE
				value := 0;
			END_IF
		END_IF
	END_IF

	// After initial interval passed, start calculating the value
	IF elapsedTime >= DINT_TO_TIME(windowS*1000) THEN
		startCalculation := TRUE;
		ready := TRUE;
	END_IF
	
END_IF
END_METHOD

END_FUNCTION_BLOCK

// ---- 01. MAIN/01.3 ReactorFlow/Handlers/01.3.2 Co2Consumption/FB_Co2ConsumptionHandler.TcPOU
FUNCTION_BLOCK FB_Co2ConsumptionHandler
VAR_INPUT
	meanFlow : REAL;
	flowControlParameters : ST_FlowControlParameters;
	resetInput : BOOL;
END_VAR
VAR_OUTPUT
	consumedCo2Amount : REAL;
	limitExceeded : BOOL;
	closeOnOffValve : BOOL;
END_VAR
VAR
	consumptionCalculator : FB_ConsumptionCalculator;
END_VAR


IF flowControlParameters.startConsumptionCalculationWithAvg THEN 
	consumptionCalculator.calculate(
								start := NOT resetInput,
								valuePerSec := meanFlow/60,
								intervalS := flowControlParameters.movingAvgShiftIntervalSecs,
								dtime := T#10MS);
END_IF
							
consumedCo2Amount := consumptionCalculator.sum;

IF resetInput THEN
	consumptionCalculator.reset();
END_IF

IF flowControlParameters.co2ConsumptionLimit > 0 AND consumedCo2Amount > flowControlParameters.co2ConsumptionLimit THEN
	limitExceeded := TRUE;
ELSE 
	limitExceeded := FALSE;
END_IF

IF flowControlParameters.closeOnOffValveIfConsumptionExceeded AND limitExceeded THEN
	closeOnOffValve := TRUE;
ELSE
	closeOnOffValve := FALSE;
END_IF

END_FUNCTION_BLOCK

// ---- 01. MAIN/01.3 ReactorFlow/FBs/FB_ConsumptionCalculator.TcPOU
FUNCTION_BLOCK FB_ConsumptionCalculator
VAR_INPUT
END_VAR
VAR_OUTPUT
	sum : REAL;
END_VAR
VAR
    running       : BOOL;
    elapsedTime   : TIME;
	RTRIG_Started : R_TRIG;
	amountOfCycles: DINT;
	counter : DINT;
END_VAR

METHOD calculate : BOOL
VAR_INPUT
	start : BOOL;
	valuePerSec : REAL;
    intervalS : INT;
    dtime : TIME;   
END_VAR
VAR
    intervalTime : TIME;
END_VAR
intervalTime := INT_TO_TIME(intervalS*1000);
RTRIG_Started(CLK := start);
// Start edge
IF RTRIG_Started.q THEN
    running := TRUE;
    sum := 0.0;
    elapsedTime := T#0S;
END_IF

IF NOT start THEN
	running := FALSE;
END_IF

IF running THEN
	// Simulate time passing
	elapsedTime := elapsedTime + dtime;
	IF elapsedTime >= intervalTime THEN
		sum := sum + valuePerSec*(intervalS);
		elapsedTime := T#0S;
		amountOfCycles := amountOfCycles + counter;
		counter := 0;
	END_IF 
	counter := counter + 1;
END_IF
END_METHOD

METHOD reset : BOOL
VAR_INPUT
END_VAR

sum := 0;
running := FALSE;
elapsedTime := T#0S;
counter := 0;
amountOfCycles := 0;
END_METHOD

END_FUNCTION_BLOCK

// ---- 01. MAIN/01.3 ReactorFlow/Handlers/01.3.3 Co2FlowModeling/FB_Co2FlowModelingHandler.TcPOU
FUNCTION_BLOCK FB_Co2FlowModelingHandler
VAR_INPUT
	valvePositionPercentage : DINT;
	pumpingPressureDelta : DINT;
	flowMeasurement : REAL;
	modelingActive : BOOL;
END_VAR
VAR_OUTPUT
	modeledOutput : LREAL;
	mF : FB_mF;
END_VAR
VAR
	u : ARRAY[1..15] OF LREAL;
	maxValveOpening : LREAL := 1.75;
	valvePosition : LREAL;
	TON_StepInterval : TON;
	firstCycle : BOOL := TRUE;
END_VAR


// Init model on first cycle
IF firstCycle THEN
	mF.setParams(
		activateObserver := TRUE);
	firstCycle := FALSE;
END_IF

// Calculate valve position
valvePosition := maxValveOpening * (TO_LREAL(valvePositionPercentage)/100);

IF modelingActive THEN
	// Fill input matrix
	u[1] := valvePosition;
	u[2] := TO_LREAL(pumpingPressureDelta);
	
	// Calculate flow every second
	TON_StepInterval(IN := TRUE, PT := T#1S);
	IF TON_StepInterval.Q THEN // AND valvePosition >= 0.25 THEN
		mF.Step(
				u := u,
				yMeas := TO_LREAL(flowMeasurement));
				
		modeledOutput := mF.y[1];
//	ELSE
//		modeledOutput := 0;
	END_IF
ELSE
	mF.Reset();
	modeledOutput := 0;
END_IF

END_FUNCTION_BLOCK

// ---- 01. MAIN/01.3 ReactorFlow/FBs/FB_mF.TcPOU
FUNCTION_BLOCK FB_mF EXTENDS FB_StateSpaceModel
VAR_INPUT
END_VAR
VAR_OUTPUT
END_VAR
VAR
END_VAR

METHOD PUBLIC setParams
VAR_INPUT
	activateObserver : BOOL;
END_VAR
VAR
    i,j : INT;
END_VAR

SUPER^();
Init(activateObserver := activateObserver);
nx := 2;
nu := 2;
ny := 1;

// Load matrices
_A[1,1] := 0.9895;
_A[1,2] := 0.03677;
_A[2,1] := -0.01237;
_A[2,2] := 0.9649;

_B[1,1] := -2.52E-05;
_B[1,2] := -1.673E-06;
_B[2,1] := -2.199E-04;
_B[2,2] := -5.346E-06;

_C[1,1] := -10.22;
_C[1,2] := -0.1235;

_K[1] := -0.1242;
_K[2] := -0.5091;
END_METHOD

END_FUNCTION_BLOCK

// ---- 01. MAIN/Common/FBs/FB_StateSpaceModel.TcPOU
FUNCTION_BLOCK ABSTRACT FB_StateSpaceModel
VAR
    nx : INT;
    nu : INT;
    ny : INT;
	
    x  		: ARRAY[1..15] OF LREAL;

    _A  : ARRAY[1..15,1..15] OF LREAL;
    _B  : ARRAY[1..15,1..15] OF LREAL;
    _C  : ARRAY[1..15,1..15] OF LREAL;
    _D  : ARRAY[1..15,1..15] OF LREAL;
    _K  : ARRAY[1..15] OF LREAL;

	_activateObserver : BOOL;
    bInit : BOOL;
	
	i,j,l : INT;
    xNext : ARRAY[1..15] OF LREAL;
    yPred : ARRAY[1..15] OF LREAL;

    e : LREAL;
END_VAR
VAR_OUTPUT
	y  : ARRAY[1..15] OF LREAL;
END_VAR

METHOD PUBLIC GetOutput
VAR_OUTPUT
    Output : ARRAY[1..15] OF LREAL;
END_VAR
VAR
    i : INT;
END_VAR

FOR i:=1 TO ny DO
    Output[i] := y[i];
END_FOR
END_METHOD

METHOD GetState
VAR_OUTPUT
    State : ARRAY[1..15] OF LREAL;
END_VAR
VAR
    i : INT;
END_VAR

FOR i:=1 TO nx DO
    State[i] := x[i];
END_FOR
END_METHOD

METHOD PUBLIC Init
VAR_INPUT
	activateObserver : BOOL;
END_VAR
VAR
    i,j : INT;
END_VAR

Reset();
//FOR i := 1 TO nx DO
//    x[i] := 0;
//    _K[i] := _K[i]; // keep
//END_FOR
_activateObserver := activateObserver;
bInit := TRUE;
END_METHOD

METHOD PUBLIC Predict
VAR_INPUT
    xIn : ARRAY[1..15] OF LREAL;
    u   : ARRAY[1..15] OF LREAL;
END_VAR
VAR_OUTPUT
    xOut : ARRAY[1..15] OF LREAL;
    yOut : ARRAY[1..15] OF LREAL;
END_VAR

(* Calculate output *)

FOR i:=1 TO ny DO

    yOut[i] := 0.0;

    FOR j:=1 TO nx DO
        yOut[i] := yOut[i] + _C[i,j] * xIn[j];
    END_FOR

    FOR j:=1 TO nu DO
        yOut[i] := yOut[i] + _D[i,j] * u[j];
    END_FOR

END_FOR


(* Predict next state *)

FOR i:=1 TO nx DO

    xOut[i] := 0.0;

    FOR j:=1 TO nx DO
        xOut[i] := xOut[i] + _A[i,j] * xIn[j];
    END_FOR

    FOR j:=1 TO nu DO
        xOut[i] := xOut[i] + _B[i,j] * u[j];
    END_FOR

END_FOR
END_METHOD

METHOD Reset : BOOL
VAR
    i : INT;
END_VAR

FOR i:=1 TO 15 DO

    x[i] := 0.0;

    y[i] := 0.0;

END_FOR
END_METHOD

METHOD setState : BOOL
VAR_INPUT
    State : ARRAY[1..15] OF LREAL;
END_VAR
VAR
    i : INT;
END_VAR

FOR i:=1 TO nx DO
    x[i] := State[i];
END_FOR
END_METHOD

METHOD PUBLIC Step
VAR_INPUT
    u      : ARRAY[1..15] OF LREAL;
    yMeas  : LREAL;
END_VAR
Predict(
    xIn := x,
    u := u,
    xOut => xNext,
    yOut => yPred);

IF _activateObserver THEN

    e := yMeas - yPred[1];

    FOR l:=1 TO nx DO
        xNext[l] := xNext[l] + _K[l] * e;
    END_FOR

END_IF

FOR l:=1 TO nx DO
    x[l] := xNext[l];
END_FOR

FOR l:=1 TO ny DO
    y[l] := yPred[l];
END_FOR
END_METHOD

END_FUNCTION_BLOCK

// ---- 01. MAIN/01.3 ReactorFlow/Handlers/01.3.4 Co2FlowModelDeviation/FB_Co2FlowModelDeviationHandler.TcPOU
FUNCTION_BLOCK FB_Co2FlowModelDeviationHandler
VAR_INPUT
	currentFlow : REAL;
	modeledFlow : REAL;
END_VAR
VAR_OUTPUT
	deviationPercentage : DINT;
END_VAR
VAR
	delta : REAL;
	_maxValue : REAL;
END_VAR


IF currentFlow <> 0 THEN
	delta := modeledFlow - currentFlow;
	
	// Normalize max value to 100 percent
	deviationPercentage := TO_DINT((delta/_maxValue)*100);
	
ELSE
	deviationPercentage := 0;
END_IF

METHOD FB_init : BOOL
VAR_INPUT
	bInitRetains : BOOL; // if TRUE, the retain variables are initialized (warm start / cold start)
	bInCopyCode : BOOL;  // if TRUE, the instance afterwards gets moved into the copy code (online change)
	maxValue : REAL;
END_VAR

_maxValue := maxValue;
END_METHOD

END_FUNCTION_BLOCK

// ---- 01. MAIN/01.3 ReactorFlow/Handlers/01.3.5 FlowMpc/FB_FlowMpcHandler.TcPOU
FUNCTION_BLOCK FB_FlowMpcHandler
VAR_INPUT
	enable : BOOL;
	flowSetpoint : REAL;
	pumpingPressureDelta : DINT;
	currentValvePosition : DINT;
	valveFullOpenTime : DINT := 25; // NOTE: Hardcoded! In the future from parameter view?
	flowModel	: FB_mF;
	measuredFlow : REAL;
END_VAR
VAR_OUTPUT
	modeledValvePercentage : DINT;
END_VAR
VAR
	maxValue : REAL := 1.75;
	currentValvePosRounds : REAL;
	valvePosRounds : REAL;

	MPC_Matrices : ST_MPC_Matrices;
	flowMpc : FB_MPC(
					MPC_Matrices := MPC_Matrices,
					PredictionHorizon := 20,
					ControlHorizon := 5);
	FlowValveLimits : ARRAY[0..1] OF REAL := [0 , 1.75];					
					
	Difference : REAL;
END_VAR


// Valve position percentage to rounds
currentValvePosRounds := (TO_REAL(currentValvePosition)/100) * maxValue;

flowMpc(
	Enable := enable,
    setpoint := flowSetpoint,
    manipulatedVariableCurrent := currentValvePosRounds,
	manipulatedVariableLimits := FlowValveLimits,
	manipulatedVariableMaxReachTime := valveFullOpenTime,
    measuredDisturbance := pumpingPressureDelta,
    controlBusy := GVL_IO.extractiveOutletControlValveClose OR GVL_IO.extractiveOutletControlValveOpen,
	measuredVariableCurrent := measuredFlow,
	Model := flowModel);

modeledValvePercentage := TO_DINT((flowMpc.ManipulatedVariableTarget / maxValue) * 100);

END_FUNCTION_BLOCK

// ---- 01. MAIN/01.3 ReactorFlow/FBs/FB_MPC.TcPOU
FUNCTION_BLOCK FB_MPC
VAR_INPUT
    enable : BOOL;

    setpoint : REAL;

